C07257=1101.391,313.700,-81.925,179.212,17.147,151.820
C07258=1101.385,313.452,-81.894,179.209,17.145,151.820
C07259=1101.379,313.204,-81.863,179.206,17.143,151.820
C07260=1101.373,312.956,-81.831,179.203,17.142,151.820
C07261=1101.368,312.708,-81.800,179.200,17.140,151.820
C07262=1101.362,312.461,-81.769,179.196,17.137,151.821
C07263=1101.356,312.212,-81.737,179.193,17.135,151.821
C07264=1101.350,311.965,-81.706,179.189,17.133,151.821
C07265=1101.345,311.716,-81.675,179.186,17.131,151.821
C07266=1101.339,311.469,-81.644,179.183,17.129,151.821
C07267=1101.333,311.221,-81.613,179.179,17.128,151.822
C07268=1101.327,310.972,-81.581,179.175,17.126,151.822
C07269=1101.322,310.725,-81.550,179.172,17.124,151.822
C07270=1101.316,310.477,-81.519,179.169,17.121,151.822
C07271=1101.310,310.229,-81.488,179.165,17.119,151.822
C07272=1101.304,309.981,-81.456,179.162,17.117,151.823
C07273=1101.299,309.733,-81.425,179.158,17.115,151.823
C07274=1101.293,309.485,-81.394,179.156,17.114,151.823
C07275=1101.288,309.237,-81.363,179.152,17.112,151.823
C07276=1101.282,308.989,-81.333,179.149,17.110,151.824
C07277=1101.276,308.741,-81.301,179.145,17.108,151.824
C07278=1101.270,308.493,-81.270,179.142,17.106,151.824
C07279=1101.265,308.245,-81.239,179.138,17.104,151.824
C07280=1101.259,307.998,-81.208,179.135,17.102,151.824
C07281=1101.253,307.749,-81.177,179.131,17.100,151.825
C07282=1101.247,307.501,-81.147,179.128,17.098,151.825
C07283=1101.242,307.254,-81.115,179.124,17.096,151.825
C07284=1101.236,307.006,-81.085,179.121,17.094,151.825
C07285=1101.230,306.757,-81.053,179.118,17.093,151.826
C07286=1101.225,306.509,-81.023,179.115,17.091,151.826
C07287=1101.219,306.262,-80.991,179.111,17.089,151.826
C07288=1101.213,306.014,-80.961,179.108,17.087,151.826
C07289=1101.208,305.766,-80.930,179.104,17.085,151.826
C07290=1101.202,305.517,-80.899,179.101,17.083,151.827
C07291=1101.197,305.269,-80.868,179.097,17.081,151.827
C07292=1101.191,305.022,-80.837,179.094,17.079,151.827
C07293=1101.186,304.774,-80.806,179.090,17.078,151.827
C07294=1101.180,304.526,-80.776,179.087,17.075,151.828
C07295=1101.174,304.277,-80.745,179.084,17.074,151.828
C07296=1101.168,304.029,-80.714,179.081,17.072,151.828
C07297=1101.162,303.781,-80.684,179.077,17.070,151.828
C07298=1101.154,303.400,-80.636,179.072,17.068,151.829
C07299=1101.146,303.018,-80.589,179.067,17.065,151.829
C07300=1101.137,302.637,-80.542,179.061,17.062,151.830
C07301=1101.128,302.254,-80.495,179.056,17.059,151.830
C07302=1101.123,302.006,-80.464,179.053,17.057,151.830
C07303=1101.117,301.758,-80.433,179.049,17.055,151.830
C07304=1101.111,301.511,-80.403,179.045,17.053,151.831
C07305=1101.106,301.262,-80.373,179.042,17.051,151.831
C07306=1101.100,301.014,-80.342,179.039,17.050,151.831
C07307=1101.095,300.766,-80.312,179.036,17.048,151.831
C07308=1101.089,300.518,-80.281,179.032,17.046,151.832
C07309=1101.084,300.270,-80.251,179.029,17.044,151.832
C07310=1101.078,300.022,-80.221,179.025,17.042,151.832
C07311=1101.073,299.774,-80.190,179.022,17.040,151.832
C07312=1101.067,299.527,-80.159,179.019,17.039,151.833
C07313=1101.061,299.278,-80.130,179.015,17.037,151.833
C07314=1101.056,299.030,-80.099,179.012,17.035,151.833
C07315=1101.051,298.782,-80.068,179.008,17.034,151.834
C07316=1101.045,298.534,-80.038,179.005,17.032,151.834
C07317=1101.039,298.286,-80.008,179.001,17.030,151.834
C07318=1101.034,298.038,-79.977,178.998,17.028,151.834
C07319=1101.028,297.790,-79.947,178.995,17.027,151.835
C07320=1101.022,297.542,-79.917,178.991,17.025,151.835
C07321=1101.017,297.294,-79.886,178.988,17.023,151.835
C07322=1101.011,297.046,-79.857,178.984,17.021,151.835
C07323=1101.005,296.798,-79.826,178.981,17.019,151.836
C07324=1101.000,296.550,-79.796,178.978,17.018,151.836
C07325=1100.994,296.302,-79.766,178.974,17.016,151.836
C07326=1100.986,295.953,-79.723,178.969,17.014,151.837
C07327=1100.978,295.604,-79.681,178.964,17.012,151.837
C07328=1100.970,295.257,-79.639,178.960,17.010,151.838
C07329=1100.961,294.908,-79.596,178.954,17.007,151.838
C07330=1100.956,294.659,-79.567,178.952,17.006,151.838
C07331=1100.950,294.412,-79.536,178.948,17.004,151.839
C07332=1100.945,294.164,-79.507,178.944,17.002,151.839
C07333=1100.939,293.916,-79.477,178.941,17.000,151.839
C07334=1100.934,293.668,-79.447,178.938,16.999,151.840
C07335=1100.928,293.420,-79.417,178.934,16.997,151.840
C07336=1100.922,293.171,-79.387,178.931,16.996,151.840
C07337=1100.917,292.924,-79.357,178.927,16.994,151.841
C07338=1100.911,292.675,-79.327,178.924,16.992,151.841
C07339=1100.905,292.427,-79.297,178.921,16.991,151.841
C07340=1100.900,292.179,-79.267,178.917,16.989,151.841
C07341=1100.894,291.931,-79.237,178.914,16.987,151.842
C07342=1100.888,291.683,-79.207,178.910,16.986,151.842
C07343=1100.883,291.434,-79.178,178.907,16.985,151.842
C07344=1100.877,291.186,-79.147,178.903,16.983,151.843
C07345=1100.872,290.938,-79.118,178.900,16.981,151.843
C07346=1100.866,290.689,-79.088,178.896,16.979,151.843
C07347=1100.860,290.442,-79.058,178.893,16.978,151.844
C07348=1100.855,290.194,-79.029,178.889,16.977,151.844
C07349=1100.849,289.946,-78.999,178.886,16.975,151.844
C07350=1100.843,289.678,-78.967,178.882,16.973,151.845
C07351=1100.837,289.410,-78.935,178.879,16.972,151.845
C07352=1100.830,289.143,-78.903,178.875,16.970,151.845
C07353=1100.824,288.875,-78.871,178.871,16.968,151.846
C07354=1100.819,288.627,-78.841,178.867,16.967,151.846
C07355=1100.814,288.379,-78.812,178.864,16.965,151.846
C07356=1100.807,288.132,-78.782,178.861,16.964,151.847
C07357=1100.802,287.883,-78.752,178.857,16.963,151.847
C07358=1100.796,287.635,-78.723,178.853,16.961,151.847
C07359=1100.790,287.387,-78.694,178.851,16.960,151.848
C07360=1100.784,287.138,-78.664,178.847,16.958,151.848
C07361=1100.779,286.890,-78.634,178.843,16.957,151.849
C07362=1100.773,286.642,-78.604,178.840,16.955,151.849
C07363=1100.767,286.394,-78.575,178.837,16.954,151.849
C07364=1100.762,286.146,-78.546,178.833,16.952,151.849
C07365=1100.756,285.898,-78.516,178.829,16.950,151.850
C07366=1100.750,285.649,-78.487,178.826,16.949,151.850
C07367=1100.745,285.401,-78.457,178.823,16.948,151.851
C07368=1100.740,285.153,-78.428,178.819,16.946,151.851
C07369=1100.733,284.905,-78.399,178.815,16.945,151.851
C07370=1100.728,284.657,-78.370,178.812,16.944,151.852
C07371=1100.722,284.408,-78.340,178.809,16.942,151.852
C07372=1100.716,284.160,-78.311,178.805,16.940,151.852
C07373=1100.711,283.912,-78.282,178.801,16.939,151.853
C07374=1100.706,283.664,-78.252,178.798,16.938,151.853
C07375=1100.699,283.416,-78.223,178.795,16.936,151.853
C07376=1100.694,283.167,-78.193,178.791,16.934,151.854
C07377=1100.688,282.920,-78.165,178.788,16.933,151.854
C07378=1100.683,282.671,-78.135,178.785,16.931,151.854
C07379=1100.678,282.422,-78.106,178.781,16.930,151.855
C07380=1100.671,282.174,-78.077,178.778,16.929,151.855
C07381=1100.666,281.927,-78.048,178.774,16.927,151.856
C07382=1100.660,281.678,-78.019,178.771,16.926,151.856
C07383=1100.655,281.430,-77.989,178.768,16.925,151.856
C07384=1100.649,281.182,-77.959,178.764,16.923,151.857
C07385=1100.644,280.933,-77.931,178.760,16.921,151.857
C07386=1100.638,280.685,-77.902,178.756,16.920,151.857
C07387=1100.632,280.437,-77.873,178.754,16.919,151.858
C07388=1100.626,280.189,-77.844,178.750,16.917,151.858
C07389=1100.621,279.941,-77.815,178.746,16.916,151.859
C07390=1100.615,279.692,-77.786,178.743,16.915,151.859
C07391=1100.609,279.444,-77.757,178.739,16.913,151.859
C07392=1100.604,279.196,-77.728,178.735,16.912,151.860
C07393=1100.599,278.947,-77.699,178.733,16.911,151.860
C07394=1100.592,278.699,-77.670,178.729,16.909,151.860
C07395=1100.587,278.452,-77.641,178.725,16.908,151.861
C07396=1100.582,278.203,-77.612,178.722,16.907,151.861
C07397=1100.575,277.955,-77.583,178.718,16.905,151.862
C07398=1100.570,277.707,-77.554,178.715,16.903,151.862
C07399=1100.564,277.458,-77.526,178.712,16.902,151.862
C07400=1100.558,277.210,-77.497,178.708,16.901,151.863
C07401=1100.554,276.962,-77.468,178.704,16.900,151.863
C07402=1100.545,276.603,-77.426,178.699,16.898,151.864
C07403=1100.537,276.244,-77.384,178.695,16.896,151.864
C07404=1100.528,275.886,-77.344,178.690,16.894,151.865
C07405=1100.520,275.528,-77.302,178.684,16.892,151.865
C07406=1100.515,275.279,-77.273,178.681,16.891,151.866
C07407=1100.509,275.031,-77.244,178.677,16.890,151.866
C07408=1100.504,274.783,-77.216,178.674,16.889,151.867
C07409=1100.498,274.534,-77.187,178.671,16.887,151.867
C07410=1100.493,274.287,-77.158,178.667,16.886,151.867
C07411=1100.487,274.038,-77.130,178.664,16.885,151.868
C07412=1100.481,273.790,-77.101,178.660,16.883,151.868
C07413=1100.475,273.542,-77.073,178.656,16.882,151.869
C07414=1100.470,273.293,-77.044,178.653,16.881,151.869
C07415=1100.464,273.045,-77.015,178.650,16.879,151.869
C07416=1100.458,272.796,-76.987,178.646,16.878,151.870
C07417=1100.452,272.548,-76.958,178.643,16.877,151.870
C07418=1100.447,272.300,-76.930,178.639,16.875,151.871
C07419=1100.441,272.052,-76.902,178.636,16.875,151.871
C07420=1100.436,271.804,-76.872,178.632,16.873,151.871
C07421=1100.430,271.555,-76.844,178.628,16.872,151.872
C07422=1100.425,271.307,-76.816,178.625,16.871,151.872
C07423=1100.419,271.058,-76.788,178.622,16.869,151.873
C07424=1100.412,270.810,-76.759,178.619,16.868,151.873
C07425=1100.407,270.562,-76.731,178.615,16.867,151.874
C07426=1100.401,270.313,-76.702,178.611,16.865,151.874
C07427=1100.397,270.065,-76.674,178.608,16.864,151.874
C07428=1100.391,269.816,-76.645,178.604,16.863,151.875
C07429=1100.385,269.569,-76.617,178.601,16.862,151.875
C07430=1100.379,269.320,-76.588,178.598,16.861,151.876
C07431=1100.374,269.072,-76.561,178.594,16.860,151.876
C07432=1100.368,268.823,-76.532,178.591,16.859,151.876
C07433=1100.362,268.575,-76.504,178.587,16.857,151.877
C07434=1100.356,268.326,-76.476,178.584,16.856,151.877
C07435=1100.351,268.078,-76.448,178.580,16.855,151.878
C07436=1100.345,267.830,-76.420,178.576,16.853,151.878
C07437=1100.340,267.582,-76.391,178.573,16.853,151.879
C07438=1100.334,267.333,-76.363,178.569,16.851,151.879
C07439=1100.328,267.085,-76.335,178.566,16.850,151.879
C07440=1100.322,266.837,-76.306,178.562,16.849,151.880
C07441=1100.317,266.589,-76.278,178.559,16.847,151.880
C07442=1100.312,266.341,-76.250,178.556,16.846,151.881
C07443=1100.306,266.092,-76.222,178.552,16.845,151.881
C07444=1100.300,265.844,-76.194,178.549,16.844,151.882
C07445=1100.294,265.595,-76.166,178.545,16.843,151.882
C07446=1100.289,265.347,-76.138,178.542,16.842,151.882
C07447=1100.283,265.098,-76.110,178.538,16.840,151.883
C07448=1100.277,264.850,-76.083,178.534,16.839,151.883
C07449=1100.272,264.602,-76.055,178.531,16.838,151.884
C07450=1100.266,264.353,-76.027,178.528,16.837,151.884
C07451=1100.261,264.105,-75.999,178.524,16.836,151.885
C07452=1100.255,263.856,-75.970,178.521,16.835,151.885
C07453=1100.249,263.608,-75.942,178.517,16.834,151.886
C07454=1100.240,263.253,-75.903,178.513,16.832,151.886
C07455=1100.232,262.897,-75.863,178.507,16.830,151.887
C07456=1100.224,262.540,-75.823,178.502,16.829,151.888
C07457=1100.216,262.185,-75.784,178.497,16.827,151.888
C07458=1100.210,261.936,-75.755,178.494,16.827,151.889
C07459=1100.205,261.688,-75.727,178.490,16.825,151.889
C07460=1100.198,261.439,-75.700,178.487,16.825,151.890
C07461=1100.193,261.191,-75.672,178.483,16.823,151.890
C07462=1100.188,260.943,-75.644,178.480,16.822,151.890
C07463=1100.181,260.695,-75.617,178.476,16.821,151.891
C07464=1100.176,260.446,-75.589,178.473,16.820,151.891
C07465=1100.171,260.198,-75.561,178.469,16.819,151.892
C07466=1100.164,259.950,-75.534,178.465,16.818,151.892
C07467=1100.159,259.701,-75.506,178.462,16.817,151.893
C07468=1100.153,259.452,-75.478,178.458,16.815,151.893
C07469=1100.147,259.205,-75.451,178.455,16.815,151.894
C07470=1100.142,258.956,-75.424,178.451,16.813,151.894
C07471=1100.136,258.707,-75.395,178.448,16.813,151.895
C07472=1100.130,258.459,-75.369,178.444,16.811,151.895
C07473=1100.125,258.211,-75.341,178.441,16.811,151.896
C07474=1100.118,257.962,-75.313,178.437,16.809,151.896
C07475=1100.113,257.714,-75.286,178.434,16.809,151.896
C07476=1100.108,257.466,-75.258,178.430,16.807,151.897
C07477=1100.102,257.217,-75.231,178.427,16.806,151.897
C07478=1100.096,256.968,-75.203,178.423,16.805,151.898
C07479=1100.090,256.720,-75.176,178.420,16.804,151.898
C07480=1100.085,256.472,-75.148,178.416,16.803,151.899
C07481=1100.079,256.223,-75.120,178.413,16.802,151.899
C07482=1100.073,255.975,-75.093,178.409,16.801,151.900
C07483=1100.068,255.726,-75.066,178.406,16.800,151.900
C07484=1100.062,255.478,-75.039,178.402,16.799,151.901
C07485=1100.056,255.229,-75.011,178.399,16.798,151.901
C07486=1100.051,254.981,-74.984,178.395,16.797,151.902
C07487=1100.045,254.733,-74.956,178.392,16.796,151.902
C07488=1100.039,254.484,-74.930,178.388,16.795,151.902
C07489=1100.034,254.235,-74.902,178.385,16.794,151.903
C07490=1100.028,253.987,-74.875,178.381,16.793,151.903
C07491=1100.023,253.739,-74.847,178.378,16.792,151.904
C07492=1100.017,253.490,-74.821,178.375,16.791,151.904
C07493=1100.012,253.242,-74.793,178.371,16.790,151.905
C07494=1100.006,252.994,-74.766,178.368,16.788,151.905
C07495=1100.000,252.744,-74.739,178.364,16.788,151.906
C07496=1099.994,252.496,-74.712,178.360,16.787,151.906
C07497=1099.989,252.248,-74.684,178.357,16.786,151.907
C07498=1099.983,252.000,-74.657,178.353,16.785,151.907
C07499=1099.978,251.751,-74.630,178.350,16.784,151.908
C07500=1099.973,251.503,-74.603,178.346,16.783,151.908
C07501=1099.967,251.253,-74.576,178.344,16.782,151.908
C07502=1099.961,251.005,-74.548,178.340,16.780,151.909
C07503=1099.956,250.757,-74.521,178.337,16.779,151.909
C07504=1099.950,250.508,-74.495,178.333,16.778,151.910
C07505=1099.945,250.260,-74.467,178.329,16.778,151.910
C07506=1099.937,249.901,-74.429,178.325,16.776,151.911
C07507=1099.929,249.543,-74.389,178.319,16.775,151.912
C07508=1099.921,249.184,-74.351,178.314,16.773,151.913
C07509=1099.913,248.825,-74.312,178.310,16.772,151.913
C07510=1099.907,248.577,-74.285,178.306,16.771,151.914
C07511=1099.902,248.329,-74.258,178.303,16.770,151.914
C07512=1099.896,248.079,-74.231,178.299,16.768,151.915
C07513=1099.890,247.831,-74.204,178.295,16.768,151.915
C07514=1099.885,247.583,-74.178,178.292,16.766,151.915
C07515=1099.879,247.334,-74.150,178.288,16.766,151.916
C07516=1099.874,247.086,-74.124,178.285,16.764,151.916
C07517=1099.868,246.837,-74.097,178.282,16.764,151.917
C07518=1099.862,246.589,-74.070,178.278,16.763,151.917
C07519=1099.857,246.340,-74.043,178.275,16.762,151.918
C07520=1099.851,246.092,-74.016,178.271,16.761,151.918
C07521=1099.846,245.843,-73.990,178.267,16.760,151.919
C07522=1099.840,245.595,-73.963,178.264,16.759,151.919
C07523=1099.835,245.346,-73.936,178.260,16.758,151.920
C07524=1099.829,245.098,-73.909,178.257,16.757,151.920
C07525=1099.823,244.850,-73.883,178.253,16.756,151.921
C07526=1099.818,244.601,-73.857,178.250,16.755,151.921
C07527=1099.812,244.352,-73.830,178.246,16.754,151.922
C07528=1099.807,244.104,-73.803,178.243,16.753,151.922
C07529=1099.801,243.855,-73.776,178.240,16.753,151.923
C07530=1099.795,243.607,-73.750,178.236,16.752,151.923
C07531=1099.790,243.358,-73.724,178.233,16.751,151.924
C07532=1099.784,243.110,-73.697,178.229,16.750,151.924
C07533=1099.778,242.861,-73.670,178.226,16.749,151.925
C07534=1099.773,242.613,-73.644,178.222,16.747,151.925
C07535=1099.767,242.364,-73.618,178.219,16.747,151.926
C07536=1099.761,242.116,-73.591,178.216,16.746,151.926
C07537=1099.756,241.867,-73.564,178.212,16.745,151.927
C07538=1099.750,241.619,-73.538,178.208,16.745,151.927
C07539=1099.744,241.370,-73.512,178.205,16.743,151.928
C07540=1099.739,241.122,-73.485,178.201,16.743,151.928
C07541=1099.733,240.873,-73.459,178.198,16.742,151.929
C07542=1099.727,240.624,-73.433,178.194,16.741,151.929
C07543=1099.722,240.376,-73.406,178.191,16.740,151.930
C07544=1099.716,240.127,-73.380,178.187,16.739,151.930
C07545=1099.710,239.878,-73.353,178.184,16.738,151.931
C07546=1099.705,239.630,-73.327,178.180,16.737,151.931
C07547=1099.699,239.381,-73.301,178.177,16.736,151.932
C07548=1099.693,239.133,-73.274,178.174,16.736,151.932
C07549=1099.688,238.884,-73.248,178.170,16.735,151.933
C07550=1099.682,238.635,-73.222,178.167,16.734,151.933
C07551=1099.677,238.386,-73.196,178.163,16.733,151.934
C07552=1099.671,238.138,-73.169,178.160,16.732,151.934
C07553=1099.665,237.889,-73.143,178.156,16.732,151.935
C07554=1099.660,237.641,-73.116,178.152,16.731,151.935
C07555=1099.654,237.392,-73.090,178.149,16.730,151.936
C07556=1099.649,237.144,-73.064,178.145,16.728,151.936
C07557=1099.643,236.895,-73.039,178.142,16.728,151.937
C07558=1099.634,236.529,-72.999,178.137,16.727,151.938
C07559=1099.626,236.164,-72.961,178.132,16.725,151.938
C07560=1099.618,235.798,-72.923,178.127,16.724,151.939
C07561=1099.610,235.433,-72.885,178.122,16.723,151.940
C07562=1099.604,235.184,-72.859,178.119,16.722,151.940
C07563=1099.598,234.936,-72.832,178.115,16.721,151.941
C07564=1099.593,234.688,-72.807,178.111,16.721,151.941
C07565=1099.587,234.439,-72.781,178.108,16.720,151.942
C07566=1099.582,234.191,-72.754,178.104,16.719,151.942
C07567=1099.576,233.942,-72.729,178.101,16.718,151.943
C07568=1099.571,233.693,-72.703,178.098,16.718,151.943
C07569=1099.564,233.444,-72.677,178.094,16.716,151.944
C07570=1099.559,233.196,-72.651,178.091,16.716,151.944
C07571=1099.554,232.947,-72.625,178.087,16.714,151.945
C07572=1099.548,232.698,-72.599,178.084,16.714,151.945
C07573=1099.542,232.450,-72.574,178.081,16.713,151.946
C07574=1099.536,232.201,-72.547,178.077,16.712,151.946
C07575=1099.532,231.953,-72.522,178.074,16.711,151.947
C07576=1099.525,231.704,-72.496,178.070,16.711,151.948
C07577=1099.520,231.455,-72.470,178.066,16.710,151.948
C07578=1099.514,231.206,-72.444,178.063,16.709,151.949
C07579=1099.509,230.959,-72.418,178.060,16.708,151.949
C07580=1099.503,230.710,-72.393,178.056,16.707,151.950
C07581=1099.498,230.461,-72.367,178.053,16.707,151.950
C07582=1099.491,230.212,-72.341,178.050,16.706,151.951
C07583=1099.486,229.963,-72.316,178.046,16.705,151.951
C07584=1099.481,229.715,-72.290,178.042,16.705,151.952
C07585=1099.475,229.467,-72.265,178.039,16.704,151.952
C07586=1099.469,229.218,-72.239,178.035,16.703,151.953
C07587=1099.463,228.969,-72.213,178.032,16.702,151.953
C07588=1099.458,228.721,-72.188,178.029,16.702,151.954
C07589=1099.452,228.472,-72.162,178.025,16.700,151.954
C07590=1099.447,228.223,-72.137,178.022,16.700,151.955
C07591=1099.440,227.974,-72.111,178.018,16.699,151.955
C07592=1099.436,227.726,-72.086,178.014,16.698,151.956
C07593=1099.429,227.477,-72.060,178.011,16.698,151.956
C07594=1099.424,227.228,-72.034,178.008,16.697,151.957
C07595=1099.418,226.980,-72.009,178.004,16.696,151.957
C07596=1099.413,226.731,-71.983,178.001,16.695,151.958
C07597=1099.407,226.483,-71.958,177.998,16.695,151.959
C07598=1099.401,226.234,-71.932,177.994,16.694,151.959
C07599=1099.395,225.986,-71.907,177.991,16.693,151.960
C07600=1099.390,225.737,-71.881,177.987,16.693,151.960
C07601=1099.384,225.488,-71.856,177.983,16.692,151.961
C07602=1099.379,225.240,-71.830,177.980,16.691,151.961
C07603=1099.373,224.991,-71.806,177.977,16.690,151.962
C07604=1099.368,224.742,-71.780,177.973,16.689,151.962
C07605=1099.362,224.494,-71.755,177.970,16.689,151.963
C07606=1099.356,224.245,-71.729,177.967,16.688,151.963
C07607=1099.351,223.997,-71.704,177.963,16.687,151.964
C07608=1099.346,223.747,-71.679,177.960,16.686,151.964
C07609=1099.340,223.498,-71.653,177.956,16.686,151.965
C07610=1099.331,223.125,-71.616,177.951,16.685,151.966
C07611=1099.323,222.751,-71.578,177.946,16.683,151.966
C07612=1099.314,222.377,-71.540,177.941,16.682,151.967
C07613=1099.306,222.003,-71.502,177.936,16.681,151.968
C07614=1099.300,221.754,-71.477,177.932,16.680,151.968
C07615=1099.295,221.506,-71.452,177.928,16.679,151.969
C07616=1099.289,221.257,-71.426,177.925,16.679,151.970
C07617=1099.283,221.008,-71.401,177.922,16.678,151.970
C07618=1099.278,220.760,-71.376,177.919,16.678,151.971
C07619=1099.272,220.510,-71.351,177.915,16.677,151.971
C07620=1099.266,220.261,-71.325,177.911,16.676,151.972
C07621=1099.261,220.014,-71.300,177.908,16.676,151.972
C07622=1099.255,219.764,-71.276,177.904,16.675,151.973
C07623=1099.249,219.516,-71.251,177.901,16.674,151.973
C07624=1099.243,219.267,-71.226,177.898,16.674,151.974
C07625=1099.238,219.019,-71.201,177.895,16.673,151.975
C07626=1099.232,218.770,-71.175,177.890,16.672,151.975
C07627=1099.227,218.521,-71.151,177.888,16.671,151.976
C07628=1099.221,218.273,-71.126,177.884,16.671,151.976
C07629=1099.215,218.023,-71.101,177.880,16.670,151.977
C07630=1099.210,217.775,-71.076,177.877,16.669,151.977
C07631=1099.204,217.526,-71.051,177.874,16.669,151.978
C07632=1099.198,217.278,-71.026,177.871,16.668,151.978
C07633=1099.193,217.029,-71.001,177.867,16.667,151.979
C07634=1099.187,216.780,-70.977,177.863,16.667,151.979
C07635=1099.182,216.531,-70.951,177.860,16.666,151.980
C07636=1099.177,216.282,-70.927,177.857,16.666,151.980
C07637=1099.170,216.034,-70.902,177.853,16.665,151.981
C07638=1099.165,215.785,-70.877,177.850,16.664,151.981
C07639=1099.159,215.536,-70.853,177.847,16.663,151.982
C07640=1099.153,215.288,-70.828,177.843,16.663,151.983
C07641=1099.148,215.039,-70.803,177.839,16.662,151.983
C07642=1099.142,214.790,-70.779,177.836,16.661,151.984
C07643=1099.137,214.542,-70.753,177.833,16.661,151.984
C07644=1099.132,214.293,-70.729,177.830,16.660,151.985
C07645=1099.126,214.044,-70.704,177.826,16.659,151.985
C07646=1099.120,213.795,-70.679,177.822,16.659,151.986
C07647=1099.115,213.547,-70.655,177.819,16.658,151.986
C07648=1099.109,213.298,-70.631,177.816,16.657,151.987
C07649=1099.103,213.049,-70.605,177.812,16.656,151.987
C07650=1099.098,212.801,-70.581,177.809,16.656,151.988
C07651=1099.092,212.552,-70.556,177.806,16.655,151.988
C07652=1099.087,212.303,-70.532,177.802,16.655,151.989
C07653=1099.081,212.054,-70.507,177.798,16.654,151.990
C07654=1099.075,211.806,-70.482,177.795,16.653,151.990
C07655=1099.070,211.557,-70.458,177.792,16.653,151.991
C07656=1099.064,211.308,-70.434,177.789,16.652,151.991
C07657=1099.059,211.059,-70.409,177.785,16.651,151.992
C07658=1099.053,210.810,-70.385,177.781,16.651,151.992
C07659=1099.047,210.562,-70.360,177.778,16.650,151.993
C07660=1099.042,210.313,-70.336,177.775,16.650,151.993
C07661=1099.035,210.064,-70.311,177.772,16.649,151.994
C07662=1099.028,209.694,-70.275,177.767,16.648,151.995
C07663=1099.019,209.324,-70.239,177.761,16.647,151.995
C07664=1099.010,208.954,-70.202,177.756,16.646,151.996
C07665=1099.002,208.584,-70.166,177.751,16.645,151.997
C07666=1098.979,207.575,-70.068,177.709,16.631,152.003
C07667=1098.974,207.326,-70.044,177.705,16.631,152.003
C07668=1098.968,207.078,-70.020,177.702,16.632,152.004
C07669=1098.963,206.829,-69.997,177.698,16.632,152.005
C07670=1098.957,206.579,-69.972,177.694,16.632,152.006
C07671=1098.951,206.331,-69.948,177.691,16.632,152.007
C07672=1098.945,206.082,-69.924,177.687,16.632,152.007
C07673=1098.940,205.834,-69.900,177.683,16.632,152.008
C07674=1098.934,205.585,-69.876,177.680,16.632,152.009
C07675=1098.928,205.336,-69.853,177.676,16.633,152.010
C07676=1098.923,205.087,-69.828,177.673,16.633,152.010
C07677=1098.918,204.839,-69.804,177.670,16.633,152.011
C07678=1098.911,204.590,-69.780,177.666,16.634,152.012
C07679=1098.906,204.340,-69.756,177.662,16.634,152.013
C07680=1098.901,204.092,-69.732,177.658,16.634,152.014
C07681=1098.895,203.843,-69.709,177.655,16.634,152.014
C07682=1098.890,203.594,-69.685,177.651,16.634,152.015
C07683=1098.883,203.345,-69.661,177.648,16.635,152.016
C07684=1098.878,203.097,-69.637,177.644,16.635,152.017
C07685=1098.873,202.848,-69.613,177.640,16.635,152.017
C07686=1098.867,202.599,-69.590,177.637,16.635,152.018
C07687=1098.862,202.351,-69.565,177.633,16.635,152.019
C07688=1098.855,202.101,-69.542,177.630,16.636,152.020
C07689=1098.850,201.852,-69.518,177.627,16.636,152.020
C07690=1098.844,201.604,-69.494,177.623,16.636,152.021
C07691=1098.838,201.355,-69.471,177.619,16.637,152.022
C07692=1098.832,201.106,-69.446,177.616,16.637,152.023
C07693=1098.826,200.858,-69.423,177.612,16.637,152.024
C07694=1098.821,200.609,-69.399,177.608,16.637,152.024
C07695=1098.815,200.360,-69.376,177.605,16.637,152.025
C07696=1098.810,200.111,-69.352,177.601,16.638,152.026
C07697=1098.804,199.862,-69.328,177.598,16.638,152.027
C07698=1098.798,199.613,-69.305,177.594,16.639,152.027
C07699=1098.793,199.365,-69.281,177.591,16.639,152.028
C07700=1098.787,199.116,-69.258,177.587,16.639,152.029
C07701=1098.781,198.867,-69.234,177.583,16.639,152.030
C07702=1098.776,198.618,-69.211,177.580,16.639,152.030
C07703=1098.769,198.369,-69.187,177.576,16.639,152.031
C07704=1098.764,198.120,-69.163,177.573,16.639,152.032
C07705=1098.758,197.872,-69.139,177.569,16.639,152.033
C07706=1098.752,197.623,-69.117,177.566,16.640,152.033
C07707=1098.747,197.374,-69.092,177.562,16.641,152.034
C07708=1098.741,197.125,-69.069,177.559,16.641,152.035
C07709=1098.736,196.876,-69.046,177.555,16.641,152.036
C07710=1098.730,196.628,-69.022,177.552,16.641,152.036
C07711=1098.725,196.379,-68.999,177.548,16.641,152.037
C07712=1098.718,196.129,-68.976,177.544,16.641,152.038
C07713=1098.713,195.881,-68.952,177.541,16.641,152.039
C07714=1098.707,195.632,-68.929,177.537,16.641,152.039
C07715=1098.701,195.383,-68.906,177.534,16.642,152.040
C07716=1098.696,195.134,-68.881,177.531,16.642,152.041
C07717=1098.690,194.885,-68.859,177.527,16.642,152.042
C07718=1098.685,194.637,-68.836,177.524,16.642,152.042
C07719=1098.679,194.388,-68.812,177.520,16.643,152.043
C07720=1098.674,194.139,-68.788,177.516,16.643,152.044
C07721=1098.668,193.890,-68.765,177.513,16.643,152.045
C07722=1098.662,193.641,-68.742,177.509,16.643,152.045
C07723=1098.657,193.393,-68.718,177.507,16.643,152.046
C07724=1098.651,193.144,-68.695,177.503,16.643,152.047
C07725=1098.645,192.895,-68.672,177.499,16.644,152.048
C07726=1098.640,192.646,-68.649,177.496,16.644,152.048
C07727=1098.633,192.373,-68.623,177.492,16.644,152.049
C07728=1098.627,192.099,-68.598,177.488,16.644,152.050
C07729=1098.621,191.825,-68.572,177.485,16.644,152.051
C07730=1098.615,191.552,-68.547,177.480,16.644,152.052
C07731=1098.610,191.303,-68.524,177.477,16.645,152.052
C07732=1098.604,191.054,-68.501,177.474,16.645,152.053
C07733=1098.599,190.805,-68.478,177.470,16.645,152.054
C07734=1098.593,190.557,-68.454,177.467,16.645,152.054
C07735=1098.588,190.307,-68.431,177.463,16.645,152.055
C07736=1098.582,190.058,-68.408,177.460,16.645,152.056
C07737=1098.576,189.810,-68.385,177.456,16.645,152.057
C07738=1098.570,189.561,-68.362,177.452,16.645,152.058
C07739=1098.565,189.312,-68.339,177.450,16.646,152.058
C07740=1098.560,189.063,-68.315,177.446,16.646,152.059
C07741=1098.554,188.814,-68.292,177.442,16.646,152.060
C07742=1098.548,188.565,-68.269,177.439,16.646,152.060
C07743=1098.543,188.316,-68.247,177.435,16.646,152.061
C07744=1098.537,188.068,-68.224,177.432,16.646,152.062
C07745=1098.532,187.819,-68.201,177.428,16.646,152.062
C07746=1098.526,187.570,-68.178,177.426,16.646,152.063
C07747=1098.521,187.321,-68.155,177.422,16.646,152.064
C07748=1098.515,187.072,-68.132,177.418,16.646,152.065
C07749=1098.509,186.823,-68.109,177.415,16.647,152.065
C07750=1098.504,186.574,-68.086,177.411,16.647,152.066
C07751=1098.498,186.325,-68.063,177.408,16.647,152.067
C07752=1098.493,186.076,-68.041,177.405,16.647,152.067
C07753=1098.487,185.827,-68.018,177.402,16.647,152.068
C07754=1098.482,185.578,-67.994,177.398,16.647,152.069
C07755=1098.477,185.329,-67.971,177.395,16.647,152.069
C07756=1098.471,185.080,-67.948,177.391,16.647,152.070
C07757=1098.465,184.832,-67.926,177.388,16.647,152.071
C07758=1098.459,184.583,-67.903,177.384,16.647,152.072
C07759=1098.453,184.333,-67.881,177.381,16.648,152.072
C07760=1098.448,184.084,-67.858,177.378,16.648,152.073
C07761=1098.443,183.836,-67.835,177.374,16.648,152.074
C07762=1098.437,183.587,-67.812,177.370,16.648,152.075
C07763=1098.430,183.339,-67.790,177.367,16.648,152.075
C07764=1098.425,183.090,-67.767,177.364,16.649,152.076
C07765=1098.419,182.840,-67.745,177.361,16.649,152.077
C07766=1098.413,182.591,-67.722,177.357,16.649,152.077
C07767=1098.408,182.343,-67.699,177.354,16.649,152.078
C07768=1098.401,182.094,-67.677,177.350,16.649,152.079
C07769=1098.396,181.844,-67.654,177.346,16.649,152.080
C07770=1098.390,181.596,-67.632,177.344,16.649,152.080
C07771=1098.385,181.347,-67.609,177.340,16.649,152.081
C07772=1098.379,181.098,-67.587,177.337,16.649,152.082
C07773=1098.373,180.849,-67.564,177.333,16.650,152.082
C07774=1098.367,180.600,-67.541,177.330,16.650,152.083
C07775=1098.362,180.351,-67.519,177.327,16.650,152.084
C07776=1098.355,180.102,-67.497,177.323,16.650,152.085
C07777=1098.350,179.853,-67.474,177.320,16.650,152.085
C07778=1098.345,179.605,-67.452,177.316,16.650,152.086
C07779=1098.339,179.356,-67.429,177.313,16.650,152.087
C07780=1098.333,179.107,-67.407,177.309,16.650,152.087
C07781=1098.327,178.858,-67.385,177.306,16.651,152.088
C07782=1098.322,178.609,-67.362,177.303,16.651,152.089
C07783=1098.317,178.360,-67.340,177.299,16.651,152.090
C07784=1098.310,178.111,-67.317,177.296,16.651,152.090
C07785=1098.305,177.862,-67.295,177.292,16.651,152.091
C07786=1098.299,177.613,-67.272,177.290,16.651,152.092
C07787=1098.293,177.364,-67.251,177.286,16.651,152.092
C07788=1098.288,177.115,-67.228,177.283,16.651,152.093
C07789=1098.282,176.866,-67.206,177.279,16.651,152.094
C07790=1098.276,176.617,-67.183,177.276,16.651,152.094
C07791=1098.270,176.343,-67.159,177.272,16.651,152.095
C07792=1098.264,176.070,-67.135,177.268,16.651,152.096
C07793=1098.258,175.795,-67.110,177.265,16.652,152.097
C07794=1098.251,175.521,-67.085,177.261,16.652,152.098
C07795=1098.246,175.272,-67.063,177.258,16.652,152.098
C07796=1098.240,175.024,-67.041,177.254,16.652,152.099
C07797=1098.234,174.774,-67.019,177.252,16.652,152.100
C07798=1098.229,174.525,-66.996,177.248,16.652,152.100
C07799=1098.224,174.277,-66.974,177.244,16.652,152.101
C07800=1098.218,174.027,-66.952,177.241,16.652,152.102
C07801=1098.212,173.779,-66.930,177.238,16.652,152.102
C07802=1098.206,173.530,-66.908,177.235,16.653,152.103
C07803=1098.201,173.281,-66.886,177.231,16.653,152.104
C07804=1098.195,173.032,-66.863,177.228,16.652,152.104
C07805=1098.190,172.783,-66.842,177.225,16.652,152.105
C07806=1098.184,172.534,-66.820,177.221,16.652,152.106
C07807=1098.178,172.285,-66.797,177.219,16.653,152.106
C07808=1098.173,172.036,-66.775,177.215,16.653,152.107
C07809=1098.167,171.787,-66.753,177.211,16.653,152.108
C07810=1098.161,171.538,-66.731,177.208,16.653,152.108
C07811=1098.156,171.289,-66.709,177.205,16.653,152.109
C07812=1098.150,171.040,-66.687,177.202,16.653,152.110
C07813=1098.145,170.791,-66.665,177.198,16.653,152.110
C07814=1098.139,170.542,-66.644,177.195,16.653,152.111
C07815=1098.133,170.293,-66.621,177.192,16.653,152.112
C07816=1098.128,170.045,-66.600,177.189,16.653,152.112
C07817=1098.122,169.795,-66.577,177.186,16.653,152.113
C07818=1098.117,169.546,-66.555,177.182,16.653,152.114
C07819=1098.111,169.297,-66.534,177.179,16.652,152.114
C07820=1098.106,169.048,-66.511,177.175,16.653,152.115
C07821=1098.100,168.800,-66.490,177.173,16.653,152.115
C07822=1098.095,168.550,-66.467,177.169,16.653,152.116
C07823=1098.089,168.302,-66.446,177.166,16.653,152.117
C07824=1098.084,168.052,-66.424,177.162,16.652,152.117
C07825=1098.078,167.804,-66.403,177.160,16.653,152.118
C07826=1098.073,167.554,-66.380,177.156,16.653,152.119
C07827=1098.067,167.306,-66.359,177.153,16.653,152.119
C07828=1098.062,167.056,-66.337,177.150,16.652,152.120
C07829=1098.055,166.807,-66.315,177.146,16.652,152.121
C07830=1098.051,166.558,-66.293,177.144,16.653,152.121
C07831=1098.044,166.309,-66.272,177.140,16.653,152.122
C07832=1098.040,166.060,-66.250,177.137,16.652,152.123
C07833=1098.033,165.811,-66.228,177.133,16.652,152.123
C07834=1098.028,165.562,-66.207,177.131,16.652,152.124
C07835=1098.022,165.313,-66.185,177.127,16.652,152.125
C07836=1098.017,165.064,-66.163,177.124,16.652,152.125
C07837=1098.012,164.816,-66.142,177.120,16.652,152.126
C07838=1098.006,164.566,-66.120,177.117,16.652,152.126
C07839=1098.001,164.318,-66.098,177.115,16.652,152.127
C07840=1097.995,164.068,-66.076,177.111,16.652,152.128
C07841=1097.990,163.820,-66.055,177.108,16.652,152.128
C07842=1097.984,163.570,-66.033,177.104,16.652,152.129
C07843=1097.978,163.322,-66.012,177.102,16.652,152.130
C07844=1097.973,163.072,-65.989,177.099,16.651,152.130
C07845=1097.967,162.824,-65.968,177.095,16.651,152.131
C07846=1097.963,162.575,-65.946,177.092,16.651,152.131
C07847=1097.957,162.325,-65.925,177.088,16.651,152.132
C07848=1097.951,162.077,-65.904,177.086,16.651,152.133
C07849=1097.946,161.827,-65.882,177.083,16.651,152.133
C07850=1097.940,161.579,-65.861,177.079,16.651,152.134
C07851=1097.934,161.329,-65.839,177.076,16.651,152.135
C07852=1097.929,161.081,-65.817,177.073,16.651,152.135
C07853=1097.923,160.831,-65.796,177.070,16.651,152.136
C07854=1097.918,160.582,-65.775,177.067,16.650,152.136
C07855=1097.911,160.308,-65.751,177.063,16.651,152.137
C07856=1097.905,160.034,-65.728,177.059,16.651,152.138
C07857=1097.899,159.759,-65.704,177.056,16.651,152.139
C07858=1097.892,159.485,-65.680,177.052,16.651,152.139
C07859=1097.887,159.236,-65.660,177.049,16.650,152.140
C07860=1097.881,158.987,-65.638,177.047,16.651,152.140
C07861=1097.875,158.738,-65.617,177.043,16.651,152.141
C07862=1097.871,158.489,-65.596,177.040,16.650,152.142
C07863=1097.865,158.239,-65.574,177.036,16.650,152.142
C07864=1097.859,157.991,-65.553,177.034,16.650,152.143
C07865=1097.853,157.741,-65.532,177.031,16.650,152.144
C07866=1097.848,157.493,-65.511,177.027,16.650,152.144
C07867=1097.842,157.244,-65.489,177.024,16.650,152.145
C07868=1097.836,156.994,-65.468,177.021,16.650,152.145
C07869=1097.831,156.746,-65.447,177.018,16.650,152.146
C07870=1097.825,156.496,-65.425,177.015,16.650,152.147
C07871=1097.820,156.247,-65.404,177.011,16.649,152.147
C07872=1097.814,155.999,-65.383,177.009,16.649,152.148
C07873=1097.809,155.749,-65.362,177.005,16.649,152.148
C07874=1097.803,155.500,-65.341,177.002,16.649,152.149
C07875=1097.797,155.251,-65.319,176.999,16.649,152.150
C07876=1097.792,155.002,-65.299,176.996,16.649,152.150
C07877=1097.786,154.753,-65.277,176.993,16.649,152.151
C07878=1097.780,154.504,-65.257,176.989,16.649,152.151
C07879=1097.775,154.255,-65.235,176.987,16.649,152.152
C07880=1097.769,154.006,-65.215,176.983,16.649,152.153
C07881=1097.763,153.757,-65.193,176.980,16.648,152.153
C07882=1097.758,153.508,-65.173,176.977,16.648,152.154
C07883=1097.752,153.259,-65.151,176.974,16.649,152.155
C07884=1097.747,153.009,-65.130,176.971,16.648,152.155
C07885=1097.741,152.761,-65.109,176.968,16.648,152.156
C07886=1097.736,152.512,-65.088,176.964,16.648,152.156
C07887=1097.730,152.263,-65.067,176.962,16.648,152.157
C07888=1097.724,152.013,-65.046,176.958,16.648,152.158
C07889=1097.719,151.764,-65.026,176.955,16.647,152.158
C07890=1097.712,151.515,-65.005,176.953,16.648,152.159
C07891=1097.707,151.266,-64.984,176.949,16.647,152.159
C07892=1097.701,151.018,-64.963,176.946,16.647,152.160
C07893=1097.696,150.769,-64.942,176.943,16.647,152.160
C07894=1097.690,150.519,-64.921,176.940,16.647,152.161
C07895=1097.685,150.270,-64.900,176.937,16.647,152.162
C07896=1097.679,150.021,-64.880,176.934,16.646,152.162
C07897=1097.674,149.771,-64.859,176.931,16.647,152.163
C07898=1097.668,149.523,-64.837,176.928,16.646,152.163
C07899=1097.663,149.274,-64.817,176.925,16.646,152.164
C07900=1097.657,149.025,-64.797,176.921,16.645,152.165
C07901=1097.651,148.776,-64.775,176.919,16.646,152.165
C07902=1097.645,148.527,-64.755,176.915,16.646,152.166
C07903=1097.640,148.277,-64.734,176.912,16.645,152.166
C07904=1097.635,148.029,-64.713,176.910,16.646,152.167
C07905=1097.628,147.779,-64.693,176.906,16.645,152.167
C07906=1097.623,147.530,-64.672,176.903,16.645,152.168
C07907=1097.617,147.281,-64.651,176.900,16.644,152.169
C07908=1097.612,147.033,-64.630,176.897,16.645,152.169
C07909=1097.605,146.783,-64.610,176.894,16.644,152.170
C07910=1097.600,146.534,-64.589,176.891,16.644,152.170
C07911=1097.595,146.285,-64.569,176.888,16.645,152.171
C07912=1097.589,146.036,-64.548,176.885,16.644,152.172
C07913=1097.583,145.787,-64.527,176.882,16.644,152.172
C07914=1097.577,145.538,-64.507,176.878,16.643,152.173
C07915=1097.572,145.289,-64.486,176.876,16.644,152.173
C07916=1097.567,145.040,-64.465,176.873,16.643,152.174
C07917=1097.561,144.791,-64.446,176.869,16.643,152.174
C07918=1097.555,144.541,-64.425,176.867,16.643,152.175
C07919=1097.549,144.267,-64.402,176.864,16.643,152.176
C07920=1097.542,143.992,-64.379,176.860,16.643,152.176
C07921=1097.537,143.718,-64.356,176.857,16.642,152.177
C07922=1097.530,143.442,-64.334,176.854,16.642,152.177
C07923=1097.525,143.193,-64.314,176.850,16.642,152.178
C07924=1097.519,142.944,-64.293,176.847,16.641,152.179
C07925=1097.513,142.695,-64.273,176.845,16.642,152.179
C07926=1097.508,142.446,-64.253,176.841,16.641,152.180
C07927=1097.503,142.197,-64.232,176.838,16.641,152.180
C07928=1097.497,141.949,-64.211,176.836,16.641,152.181
C07929=1097.491,141.699,-64.191,176.832,16.641,152.181
C07930=1097.485,141.450,-64.170,176.829,16.640,152.182
C07931=1097.480,141.200,-64.151,176.827,16.640,152.183
C07932=1097.474,140.951,-64.130,176.824,16.640,152.183
C07933=1097.469,140.703,-64.110,176.820,16.639,152.184
C07934=1097.463,140.453,-64.090,176.817,16.639,152.184
C07935=1097.458,140.204,-64.069,176.815,16.639,152.185
C07936=1097.452,139.955,-64.049,176.811,16.639,152.185
C07937=1097.446,139.706,-64.028,176.808,16.638,152.186
C07938=1097.440,139.457,-64.008,176.806,16.639,152.186
C07939=1097.435,139.208,-63.988,176.802,16.638,152.187
C07940=1097.429,138.959,-63.968,176.799,16.638,152.187
C07941=1097.424,138.710,-63.947,176.797,16.638,152.188
C07942=1097.418,138.461,-63.927,176.794,16.637,152.188
C07943=1097.412,138.212,-63.907,176.790,16.637,152.189
C07944=1097.407,137.962,-63.887,176.788,16.637,152.190
C07945=1097.401,137.713,-63.867,176.785,16.637,152.190
C07946=1097.395,137.464,-63.847,176.781,16.636,152.191
C07947=1097.390,137.215,-63.826,176.779,16.637,152.191
C07948=1097.384,136.966,-63.806,176.776,16.636,152.192
C07949=1097.378,136.717,-63.786,176.773,16.635,152.192
C07950=1097.373,136.467,-63.766,176.770,16.636,152.193
C07951=1097.367,136.218,-63.746,176.767,16.635,152.193
C07952=1097.361,135.969,-63.726,176.764,16.635,152.194
C07953=1097.355,135.721,-63.706,176.762,16.635,152.194
C07954=1097.350,135.471,-63.686,176.758,16.634,152.195
C07955=1097.344,135.222,-63.666,176.755,16.634,152.196
C07956=1097.339,134.973,-63.645,176.753,16.634,152.196
C07957=1097.333,134.724,-63.626,176.750,16.633,152.196
C07958=1097.328,134.474,-63.606,176.746,16.633,152.197
C07959=1097.322,134.225,-63.586,176.744,16.633,152.198
C07960=1097.316,133.977,-63.566,176.741,16.633,152.198
C07961=1097.311,133.727,-63.546,176.738,16.632,152.199
C07962=1097.305,133.478,-63.526,176.735,16.632,152.199
C07963=1097.300,133.229,-63.505,176.732,16.632,152.200
C07964=1097.294,132.980,-63.486,176.729,16.631,152.200
C07965=1097.288,132.731,-63.466,176.726,16.631,152.201
C07966=1097.283,132.482,-63.446,176.723,16.631,152.201
C07967=1097.277,132.232,-63.426,176.720,16.630,152.202
C07968=1097.271,131.983,-63.406,176.718,16.630,152.202
C07969=1097.265,131.735,-63.386,176.715,16.630,152.203
C07970=1097.261,131.485,-63.367,176.711,16.629,152.203
C07971=1097.255,131.236,-63.347,176.709,16.629,152.204
C07972=1097.249,130.987,-63.327,176.706,16.629,152.204
C07973=1097.243,130.738,-63.308,176.703,16.628,152.205
C07974=1097.237,130.488,-63.288,176.700,16.629,152.205
C07975=1097.232,130.239,-63.268,176.697,16.628,152.206
C07976=1097.226,129.990,-63.248,176.694,16.628,152.206
C07977=1097.220,129.741,-63.229,176.691,16.628,152.207
C07978=1097.214,129.492,-63.209,176.688,16.627,152.207
C07979=1097.209,129.243,-63.189,176.685,16.627,152.208
C07980=1097.203,128.994,-63.169,176.683,16.627,152.209
C07981=1097.198,128.744,-63.150,176.680,16.626,152.209
C07982=1097.192,128.495,-63.130,176.676,16.626,152.210
C07983=1097.185,128.221,-63.108,176.674,16.626,152.210
C07984=1097.179,127.945,-63.086,176.671,16.625,152.211
C07985=1097.173,127.671,-63.065,176.667,16.625,152.211
C07986=1097.167,127.396,-63.043,176.664,16.625,152.212
C07987=1097.161,127.147,-63.024,176.661,16.624,152.212
C07988=1097.155,126.898,-63.004,176.658,16.624,152.213
C07989=1097.149,126.649,-62.985,176.656,16.623,152.213
C07990=1097.144,126.399,-62.965,176.652,16.623,152.214
C07991=1097.138,126.150,-62.945,176.650,16.623,152.214
C07992=1097.133,125.901,-62.925,176.647,16.622,152.215
C07993=1097.127,125.651,-62.906,176.644,16.622,152.215
C07994=1097.121,125.402,-62.886,176.642,16.622,152.216
C07995=1097.115,125.153,-62.867,176.639,16.621,152.216
C07996=1097.110,124.904,-62.848,176.635,16.621,152.217
C07997=1097.104,124.655,-62.828,176.633,16.621,152.217
C07998=1097.098,124.406,-62.809,176.630,16.620,152.218
C07999=1097.093,124.157,-62.790,176.627,16.619,152.218
C08000=1097.087,123.908,-62.770,176.624,16.619,152.219
C08001=1097.081,123.658,-62.751,176.621,16.619,152.219
C08002=1097.075,123.409,-62.731,176.619,16.619,152.220
C08003=1097.071,123.160,-62.711,176.616,16.618,152.220
C08004=1097.065,122.911,-62.692,176.613,16.618,152.221
C08005=1097.059,122.662,-62.673,176.611,16.617,152.221
C08006=1097.054,122.412,-62.653,176.607,16.617,152.222
C08007=1097.048,122.163,-62.633,176.604,16.616,152.222
C08008=1097.042,121.914,-62.614,176.602,16.616,152.223
C08009=1097.037,121.665,-62.595,176.599,16.616,152.223
C08010=1097.031,121.416,-62.576,176.596,16.615,152.224
C08011=1097.026,121.166,-62.557,176.593,16.615,152.224
C08012=1097.020,120.917,-62.538,176.591,16.614,152.224
C08013=1097.014,120.668,-62.518,176.588,16.614,152.225
C08014=1097.009,120.419,-62.499,176.585,16.614,152.225
C08015=1097.003,120.170,-62.479,176.582,16.613,152.226
C08016=1096.997,119.920,-62.460,176.580,16.613,152.226
C08017=1096.992,119.671,-62.441,176.577,16.612,152.227
C08018=1096.986,119.422,-62.422,176.574,16.611,152.227
C08019=1096.981,119.173,-62.403,176.571,16.611,152.228
C08020=1096.975,118.924,-62.383,176.568,16.611,152.228
C08021=1096.969,118.675,-62.364,176.566,16.611,152.229
C08022=1096.964,118.425,-62.344,176.563,16.610,152.229
C08023=1096.958,118.176,-62.326,176.560,16.609,152.229
C08024=1096.953,117.927,-62.306,176.558,16.609,152.230
C08025=1096.947,117.678,-62.287,176.555,16.608,152.230
C08026=1096.942,117.429,-62.268,176.552,16.608,152.231
C08027=1096.936,117.179,-62.249,176.549,16.608,152.231
C08028=1096.931,116.930,-62.230,176.546,16.607,152.232
C08029=1096.925,116.681,-62.210,176.544,16.607,152.232
C08030=1096.920,116.432,-62.192,176.541,16.606,152.233
C08031=1096.913,116.183,-62.173,176.538,16.605,152.233
C08032=1096.908,115.933,-62.154,176.536,16.605,152.234
C08033=1096.903,115.685,-62.135,176.533,16.605,152.234
C08034=1096.897,115.435,-62.116,176.530,16.604,152.234
C08035=1096.891,115.186,-62.096,176.527,16.604,152.235
C08036=1096.886,114.937,-62.077,176.525,16.603,152.235
C08037=1096.880,114.688,-62.058,176.522,16.602,152.236
C08038=1096.875,114.438,-62.039,176.519,16.602,152.236
C08039=1096.870,114.189,-62.021,176.516,16.601,152.237
C08040=1096.864,113.940,-62.002,176.514,16.601,152.237
C08041=1096.858,113.690,-61.983,176.511,16.600,152.238
C08042=1096.852,113.441,-61.964,176.509,16.600,152.238
C08043=1096.847,113.192,-61.945,176.505,16.600,152.239
C08044=1096.841,112.943,-61.926,176.503,16.599,152.239
C08045=1096.835,112.693,-61.907,176.500,16.599,152.239
C08046=1096.830,112.445,-61.888,176.497,16.598,152.240
C08047=1096.824,112.170,-61.867,176.494,16.598,152.240
C08048=1096.818,111.895,-61.847,176.492,16.597,152.241
C08049=1096.811,111.620,-61.825,176.489,16.596,152.241
C08050=1096.805,111.345,-61.805,176.486,16.596,152.242
C08051=1096.799,111.096,-61.786,176.483,16.595,152.242
C08052=1096.793,110.847,-61.768,176.481,16.595,152.243
C08053=1096.788,110.597,-61.749,176.478,16.594,152.243
C08054=1096.782,110.348,-61.730,176.475,16.593,152.243
C08055=1096.777,110.099,-61.712,176.472,16.594,152.244
C08056=1096.771,109.850,-61.692,176.469,16.593,152.244
C08057=1096.765,109.600,-61.674,176.467,16.593,152.245
C08058=1096.760,109.351,-61.656,176.464,16.592,152.245
C08059=1096.754,109.102,-61.636,176.461,16.591,152.246
C08060=1096.748,108.853,-61.618,176.459,16.591,152.246
C08061=1096.743,108.604,-61.599,176.456,16.590,152.247
C08062=1096.737,108.354,-61.580,176.454,16.590,152.247
C08063=1096.731,108.105,-61.562,176.451,16.589,152.247
C08064=1096.726,107.856,-61.543,176.448,16.588,152.248
C08065=1096.719,107.607,-61.525,176.445,16.588,152.248
C08066=1096.714,107.358,-61.506,176.442,16.588,152.249
C08067=1096.709,107.108,-61.487,176.440,16.587,152.249
C08068=1096.703,106.859,-61.469,176.437,16.587,152.250
C08069=1096.698,106.609,-61.451,176.435,16.586,152.250
C08070=1096.691,106.360,-61.432,176.432,16.586,152.250
C08071=1096.686,106.111,-61.413,176.429,16.585,152.251
C08072=1096.680,105.862,-61.395,176.427,16.584,152.251
C08073=1096.674,105.612,-61.376,176.424,16.584,152.252
C08074=1096.670,105.363,-61.358,176.422,16.583,152.252
C08075=1096.663,105.114,-61.339,176.419,16.583,152.252
C08076=1096.658,104.865,-61.320,176.416,16.582,152.253
C08077=1096.652,104.615,-61.302,176.413,16.582,152.253
C08078=1096.647,104.367,-61.283,176.410,16.581,152.254
C08079=1096.641,104.117,-61.265,176.409,16.580,152.254
C08080=1096.636,103.868,-61.247,176.406,16.579,152.254
C08081=1096.630,103.618,-61.229,176.403,16.579,152.255
C08082=1096.624,103.370,-61.210,176.400,16.578,152.255
C08083=1096.618,103.120,-61.192,176.397,16.577,152.256
C08084=1096.613,102.871,-61.173,176.395,16.577,152.256
C08085=1096.607,102.621,-61.155,176.392,16.576,152.256
C08086=1096.602,102.373,-61.136,176.390,16.576,152.257
C08087=1096.596,102.123,-61.118,176.387,16.575,152.257
C08088=1096.591,101.874,-61.099,176.385,16.575,152.258
C08089=1096.585,101.624,-61.081,176.382,16.574,152.258
C08090=1096.580,101.375,-61.063,176.379,16.573,152.258
C08091=1096.574,101.126,-61.045,176.377,16.573,152.259
C08092=1096.569,100.877,-61.026,176.374,16.572,152.259
C08093=1096.562,100.628,-61.008,176.372,16.572,152.260
C08094=1096.556,100.378,-60.990,176.369,16.571,152.260
C08095=1096.551,100.128,-60.972,176.367,16.571,152.260
C08096=1096.545,99.879,-60.953,176.364,16.570,152.261
C08097=1096.540,99.630,-60.935,176.361,16.569,152.261
C08098=1096.534,99.381,-60.916,176.359,16.569,152.262
C08099=1096.528,99.132,-60.899,176.356,16.568,152.262
C08100=1096.522,98.882,-60.881,176.354,16.567,152.262
C08101=1096.516,98.634,-60.862,176.351,16.567,152.263
C08102=1096.511,98.384,-60.844,176.349,16.566,152.263
C08103=1096.505,98.135,-60.826,176.346,16.566,152.264
C08104=1096.500,97.885,-60.809,176.343,16.565,152.264
C08105=1096.494,97.636,-60.789,176.341,16.564,152.264
C08106=1096.489,97.387,-60.772,176.338,16.563,152.265
C08107=1096.483,97.137,-60.754,176.336,16.563,152.265
C08108=1096.478,96.889,-60.735,176.333,16.562,152.266
C08109=1096.471,96.639,-60.717,176.330,16.562,152.266
C08110=1096.466,96.390,-60.700,176.328,16.561,152.266
C08111=1096.459,96.115,-60.679,176.325,16.560,152.267
C08112=1096.453,95.841,-60.660,176.323,16.560,152.267
C08113=1096.447,95.565,-60.640,176.320,16.559,152.267
C08114=1096.441,95.291,-60.620,176.317,16.558,152.268
C08115=1096.435,95.041,-60.602,176.314,16.557,152.268
C08116=1096.430,94.792,-60.584,176.311,16.557,152.269
C08117=1096.424,94.543,-60.565,176.309,16.556,152.269
C08118=1096.418,94.294,-60.548,176.307,16.556,152.269
C08119=1096.413,94.045,-60.530,176.304,16.555,152.270
C08120=1096.407,93.795,-60.512,176.302,16.554,152.270
C08121=1096.402,93.546,-60.494,176.299,16.553,152.271
C08122=1096.396,93.296,-60.476,176.297,16.553,152.271
C08123=1096.390,93.047,-60.459,176.294,16.552,152.271
C08124=1096.384,92.798,-60.440,176.292,16.552,152.272
C08125=1096.379,92.548,-60.422,176.289,16.551,152.272
C08126=1096.374,92.299,-60.404,176.286,16.550,152.272
C08127=1096.368,92.050,-60.387,176.284,16.549,152.273
C08128=1096.362,91.801,-60.369,176.281,16.549,152.273
C08129=1096.356,91.551,-60.351,176.279,16.548,152.273
C08130=1096.352,91.302,-60.333,176.276,16.547,152.274
C08131=1096.346,91.052,-60.315,176.274,16.546,152.274
C08132=1096.340,90.803,-60.298,176.271,16.546,152.274
C08133=1096.334,90.554,-60.280,176.269,16.545,152.275
C08134=1096.328,90.305,-60.262,176.266,16.544,152.275
C08135=1096.323,90.056,-60.244,176.264,16.544,152.276
C08136=1096.317,89.806,-60.227,176.261,16.543,152.276
C08137=1096.311,89.557,-60.209,176.259,16.542,152.276
C08138=1096.306,89.308,-60.191,176.256,16.542,152.277
C08139=1096.300,89.058,-60.173,176.253,16.541,152.277
C08140=1096.294,88.809,-60.156,176.251,16.540,152.277
C08141=1096.289,88.560,-60.138,176.248,16.539,152.278
C08142=1096.282,88.310,-60.120,176.246,16.539,152.278
C08143=1096.277,88.061,-60.103,176.243,16.538,152.278
C08144=1096.271,87.812,-60.085,176.241,16.538,152.279
C08145=1096.265,87.562,-60.067,176.239,16.536,152.279
C08146=1096.260,87.313,-60.050,176.236,16.536,152.280
C08147=1096.254,87.064,-60.032,176.233,16.535,152.280
C08148=1096.248,86.814,-60.015,176.232,16.535,152.280
C08149=1096.243,86.565,-59.997,176.229,16.534,152.281
C08150=1096.237,86.316,-59.980,176.227,16.533,152.281
C08151=1096.231,86.066,-59.962,176.224,16.532,152.281
C08152=1096.226,85.817,-59.944,176.222,16.532,152.282
C08153=1096.220,85.568,-59.927,176.219,16.531,152.282
C08154=1096.215,85.319,-59.909,176.217,16.530,152.282
C08155=1096.209,85.069,-59.892,176.214,16.529,152.283
C08156=1096.203,84.820,-59.874,176.212,16.529,152.283
C08157=1096.198,84.570,-59.857,176.209,16.528,152.283
C08158=1096.192,84.321,-59.839,176.207,16.527,152.284
C08159=1096.185,84.072,-59.822,176.204,16.526,152.284
C08160=1096.180,83.822,-59.805,176.202,16.525,152.284
C08161=1096.175,83.573,-59.788,176.199,16.525,152.285
C08162=1096.169,83.324,-59.770,176.197,16.524,152.285
C08163=1096.163,83.075,-59.752,176.194,16.523,152.285
C08164=1096.158,82.825,-59.734,176.192,16.522,152.286
C08165=1096.152,82.576,-59.718,176.190,16.522,152.286
C08166=1096.147,82.327,-59.700,176.187,16.521,152.286
C08167=1096.141,82.077,-59.682,176.185,16.520,152.287
C08168=1096.136,81.827,-59.665,176.182,16.519,152.287
C08169=1096.130,81.578,-59.648,176.180,16.519,152.287
C08170=1096.124,81.329,-59.630,176.177,16.518,152.288
C08171=1096.119,81.080,-59.614,176.175,16.517,152.288
C08172=1096.112,80.830,-59.596,176.173,16.516,152.288
C08173=1096.107,80.581,-59.578,176.170,16.516,152.289
C08174=1096.102,80.332,-59.562,176.168,16.514,152.289
C08175=1096.096,80.057,-59.542,176.165,16.514,152.289
C08176=1096.089,79.783,-59.523,176.163,16.513,152.290
C08177=1096.084,79.508,-59.504,176.160,16.512,152.290
C08178=1096.077,79.233,-59.485,176.157,16.511,152.290
C08179=1096.071,78.984,-59.467,176.155,16.510,152.290
C08180=1096.066,78.734,-59.451,176.152,16.509,152.291
C08181=1096.060,78.485,-59.434,176.150,16.509,152.291
C08182=1096.055,78.236,-59.417,176.147,16.508,152.292
C08183=1096.048,77.986,-59.399,176.145,16.507,152.292
C08184=1096.043,77.737,-59.381,176.143,16.506,152.292
C08185=1096.037,77.488,-59.365,176.141,16.506,152.293
C08186=1096.031,77.239,-59.347,176.138,16.504,152.293
C08187=1096.026,76.989,-59.331,176.136,16.504,152.293
C08188=1096.020,76.740,-59.314,176.133,16.503,152.293
C08189=1096.014,76.490,-59.296,176.131,16.502,152.294
C08190=1096.009,76.241,-59.279,176.128,16.501,152.294
C08191=1096.003,75.991,-59.262,176.126,16.501,152.294
C08192=1095.997,75.742,-59.245,176.124,16.499,152.295
C08193=1095.992,75.493,-59.228,176.122,16.499,152.295
C08194=1095.986,75.244,-59.211,176.119,16.498,152.295
C08195=1095.980,74.994,-59.194,176.117,16.497,152.296
C08196=1095.974,74.745,-59.176,176.114,16.496,152.296
C08197=1095.968,74.495,-59.160,176.112,16.495,152.296
C08198=1095.963,74.246,-59.143,176.109,16.495,152.297
C08199=1095.958,73.997,-59.126,176.107,16.494,152.297
C08200=1095.952,73.747,-59.109,176.105,16.493,152.297
C08201=1095.946,73.498,-59.092,176.103,16.492,152.297
C08202=1095.941,73.248,-59.075,176.100,16.491,152.298
C08203=1095.935,73.000,-59.058,176.098,16.490,152.298
C08204=1095.930,72.750,-59.041,176.095,16.489,152.298
C08205=1095.924,72.500,-59.024,176.093,16.489,152.299
C08206=1095.918,72.252,-59.007,176.091,16.488,152.299
C08207=1095.912,72.001,-58.990,176.088,16.487,152.299
C08208=1095.906,71.752,-58.974,176.087,16.486,152.299
C08209=1095.901,71.503,-58.956,176.084,16.485,152.300
C08210=1095.896,71.253,-58.940,176.082,16.484,152.300
C08211=1095.890,71.004,-58.923,176.079,16.484,152.300
C08212=1095.884,70.755,-58.906,176.077,16.483,152.301
C08213=1095.878,70.506,-58.889,176.074,16.482,152.301
C08214=1095.873,70.256,-58.873,176.072,16.481,152.301
C08215=1095.867,70.007,-58.856,176.070,16.480,152.301
C08216=1095.861,69.758,-58.839,176.068,16.479,152.302
C08217=1095.856,69.508,-58.822,176.065,16.478,152.302
C08218=1095.850,69.259,-58.806,176.063,16.478,152.302
C08219=1095.844,69.010,-58.789,176.060,16.476,152.303
C08220=1095.839,68.760,-58.772,176.058,16.476,152.303
C08221=1095.833,68.511,-58.756,176.056,16.474,152.303
C08222=1095.828,68.261,-58.739,176.054,16.474,152.303
C08223=1095.821,68.012,-58.722,176.051,16.473,152.304
C08224=1095.816,67.763,-58.705,176.049,16.472,152.304
C08225=1095.810,67.513,-58.689,176.047,16.472,152.304
C08226=1095.805,67.264,-58.672,176.044,16.470,152.305
C08227=1095.799,67.014,-58.656,176.042,16.470,152.305
C08228=1095.794,66.765,-58.638,176.040,16.468,152.305
C08229=1095.788,66.516,-58.622,176.038,16.468,152.305
C08230=1095.782,66.267,-58.605,176.035,16.467,152.306
C08231=1095.776,66.017,-58.589,176.033,16.466,152.306
C08232=1095.770,65.768,-58.572,176.030,16.465,152.306
C08233=1095.765,65.518,-58.555,176.028,16.464,152.307
C08234=1095.759,65.269,-58.539,176.026,16.463,152.307
C08235=1095.753,65.020,-58.522,176.024,16.462,152.307
C08236=1095.748,64.770,-58.505,176.021,16.461,152.307
C08237=1095.742,64.521,-58.489,176.019,16.460,152.308
C08238=1095.737,64.271,-58.472,176.017,16.460,152.308
C08239=1095.730,63.997,-58.454,176.014,16.459,152.308
C08240=1095.724,63.722,-58.436,176.012,16.458,152.309
C08241=1095.717,63.447,-58.418,176.009,16.456,152.309
C08242=1095.710,63.172,-58.400,176.007,16.456,152.309
C08243=1095.705,62.922,-58.383,176.004,16.454,152.310
C08244=1095.699,62.673,-58.367,176.003,16.454,152.310
C08245=1095.693,62.424,-58.351,176.000,16.453,152.310
C08246=1095.687,62.174,-58.334,175.998,16.452,152.310
C08247=1095.681,61.925,-58.318,175.996,16.452,152.311
C08248=1095.676,61.675,-58.302,175.993,16.450,152.311
C08249=1095.670,61.426,-58.285,175.991,16.450,152.311
C08250=1095.664,61.176,-58.268,175.988,16.448,152.311
C08251=1095.659,60.928,-58.253,175.987,16.448,152.312
C08252=1095.653,60.678,-58.236,175.984,16.446,152.312
C08253=1095.647,60.429,-58.220,175.982,16.446,152.312
C08254=1095.641,60.179,-58.204,175.979,16.444,152.313
C08255=1095.636,59.930,-58.187,175.977,16.444,152.313
C08256=1095.630,59.680,-58.171,175.976,16.443,152.313
C08257=1095.624,59.431,-58.154,175.973,16.442,152.313
C08258=1095.618,59.182,-58.138,175.971,16.441,152.314
C08259=1095.612,58.932,-58.122,175.968,16.440,152.314
C08260=1095.606,58.683,-58.106,175.966,16.439,152.314
C08261=1095.601,58.433,-58.089,175.964,16.438,152.314
C08262=1095.595,58.184,-58.073,175.962,16.437,152.315
C08263=1095.589,57.934,-58.057,175.960,16.437,152.315
C08264=1095.583,57.685,-58.041,175.957,16.435,152.315
C08265=1095.577,57.435,-58.025,175.955,16.435,152.315
C08266=1095.572,57.187,-58.009,175.953,16.433,152.316
C08267=1095.566,56.937,-57.992,175.951,16.433,152.316
C08268=1095.561,56.688,-57.976,175.948,16.431,152.316
C08269=1095.555,56.438,-57.959,175.946,16.431,152.316
C08270=1095.549,56.188,-57.944,175.944,16.430,152.317
C08271=1095.543,55.939,-57.927,175.941,16.429,152.317
C08272=1095.537,55.690,-57.911,175.940,16.428,152.317
C08273=1095.531,55.440,-57.895,175.937,16.427,152.318
C08274=1095.526,55.192,-57.879,175.935,16.426,152.318
C08275=1095.520,54.942,-57.864,175.933,16.424,152.318
C08276=1095.515,54.692,-57.847,175.931,16.424,152.318
C08277=1095.509,54.443,-57.830,175.929,16.423,152.318
C08278=1095.503,54.193,-57.814,175.926,16.422,152.319
C08279=1095.498,53.943,-57.799,175.924,16.421,152.319
C08280=1095.492,53.695,-57.783,175.922,16.420,152.319
C08281=1095.486,53.445,-57.766,175.920,16.419,152.319
C08282=1095.481,53.195,-57.751,175.917,16.418,152.320
C08283=1095.475,52.946,-57.735,175.915,16.417,152.320
C08284=1095.469,52.697,-57.718,175.913,16.416,152.320
C08285=1095.464,52.448,-57.703,175.911,16.415,152.320
C08286=1095.458,52.198,-57.687,175.909,16.414,152.321
C08287=1095.452,51.949,-57.671,175.906,16.413,152.321
C08288=1095.446,51.699,-57.654,175.904,16.412,152.321
C08289=1095.440,51.450,-57.639,175.903,16.411,152.321
C08290=1095.436,51.201,-57.622,175.900,16.410,152.322
C08291=1095.430,50.951,-57.607,175.898,16.409,152.322
C08292=1095.424,50.701,-57.591,175.895,16.408,152.322
C08293=1095.418,50.452,-57.574,175.894,16.407,152.322
C08294=1095.413,50.203,-57.559,175.891,16.405,152.322
C08295=1095.407,49.953,-57.543,175.889,16.405,152.323
C08296=1095.402,49.703,-57.527,175.887,16.404,152.323
C08297=1095.396,49.454,-57.511,175.885,16.403,152.323
C08298=1095.390,49.205,-57.495,175.883,16.402,152.323
C08299=1095.385,48.955,-57.480,175.880,16.400,152.324
C08300=1095.379,48.706,-57.463,175.878,16.400,152.324
C08301=1095.373,48.456,-57.448,175.877,16.399,152.324
C08302=1095.368,48.207,-57.432,175.874,16.397,152.324
C08303=1095.361,47.933,-57.415,175.872,16.397,152.324
C08304=1095.355,47.657,-57.398,175.870,16.395,152.325
C08305=1095.349,47.382,-57.380,175.867,16.394,152.325
C08306=1095.342,47.107,-57.363,175.865,16.393,152.325
C08307=1095.337,46.858,-57.347,175.863,16.392,152.325
C08308=1095.331,46.608,-57.331,175.861,16.391,152.326
C08309=1095.326,46.358,-57.316,175.858,16.390,152.326
C08310=1095.320,46.110,-57.300,175.856,16.389,152.326
C08311=1095.315,45.860,-57.284,175.854,16.388,152.326
C08312=1095.309,45.610,-57.268,175.852,16.387,152.327
C08313=1095.304,45.361,-57.253,175.850,16.385,152.327
C08314=1095.298,45.112,-57.236,175.847,16.384,152.327
C08315=1095.292,44.862,-57.221,175.846,16.384,152.327
C08316=1095.287,44.613,-57.205,175.844,16.382,152.327
C08317=1095.281,44.363,-57.189,175.841,16.381,152.328
C08318=1095.275,44.113,-57.174,175.839,16.380,152.328
C08319=1095.270,43.865,-57.158,175.837,16.379,152.328
C08320=1095.264,43.615,-57.143,175.835,16.378,152.328
C08321=1095.258,43.366,-57.127,175.833,16.377,152.328
C08322=1095.253,43.116,-57.112,175.831,16.376,152.329
C08323=1095.247,42.866,-57.096,175.829,16.375,152.329
C08324=1095.241,42.617,-57.080,175.826,16.374,152.329
C08325=1095.235,42.368,-57.065,175.825,16.372,152.329
C08326=1095.230,42.118,-57.050,175.823,16.372,152.329
C08327=1095.224,41.869,-57.034,175.820,16.371,152.330
C08328=1095.219,41.619,-57.018,175.818,16.369,152.330
C08329=1095.213,41.369,-57.003,175.817,16.369,152.330
C08330=1095.206,41.120,-56.987,175.814,16.367,152.330
C08331=1095.201,40.871,-56.972,175.812,16.366,152.330
C08332=1095.196,40.621,-56.956,175.810,16.365,152.331
C08333=1095.191,40.372,-56.941,175.808,16.364,152.331
C08334=1095.184,40.123,-56.926,175.806,16.363,152.331
C08335=1095.178,39.873,-56.910,175.803,16.362,152.331
C08336=1095.173,39.624,-56.895,175.801,16.361,152.332
C08337=1095.167,39.374,-56.879,175.800,16.360,152.332
C08338=1095.161,39.125,-56.864,175.797,16.359,152.332
C08339=1095.156,38.875,-56.848,175.796,16.358,152.332
C08340=1095.150,38.625,-56.833,175.793,16.356,152.332
C08341=1095.145,38.376,-56.818,175.791,16.356,152.333
C08342=1095.138,38.127,-56.802,175.789,16.355,152.333
C08343=1095.133,37.878,-56.787,175.787,16.353,152.333
C08344=1095.128,37.628,-56.771,175.785,16.352,152.333
C08345=1095.121,37.378,-56.756,175.783,16.351,152.333
C08346=1095.116,37.129,-56.741,175.780,16.350,152.334
C08347=1095.110,36.880,-56.726,175.779,16.349,152.334
C08348=1095.104,36.630,-56.710,175.776,16.348,152.334
C08349=1095.099,36.381,-56.695,175.774,16.347,152.334
C08350=1095.093,36.131,-56.680,175.773,16.346,152.334
C08351=1095.087,35.882,-56.665,175.770,16.345,152.335
C08352=1095.081,35.632,-56.650,175.768,16.344,152.335
C08353=1095.075,35.382,-56.634,175.766,16.343,152.335
C08354=1095.069,35.134,-56.619,175.764,16.342,152.335
C08355=1095.064,34.884,-56.603,175.762,16.340,152.335
C08356=1095.058,34.635,-56.589,175.760,16.340,152.336
C08357=1095.052,34.385,-56.573,175.758,16.338,152.336
C08358=1095.047,34.136,-56.558,175.756,16.337,152.336
C08359=1095.041,33.886,-56.543,175.754,16.337,152.336
C08360=1095.035,33.636,-56.528,175.752,16.335,152.336
C08361=1095.029,33.387,-56.513,175.750,16.334,152.337
C08362=1095.024,33.137,-56.498,175.748,16.333,152.337
C08363=1095.018,32.888,-56.483,175.746,16.332,152.337
C08364=1095.012,32.638,-56.467,175.744,16.331,152.337
C08365=1095.007,32.389,-56.453,175.741,16.329,152.337
C08366=1095.001,32.139,-56.437,175.740,16.328,152.338
C08367=1094.995,31.865,-56.420,175.738,16.328,152.338
C08368=1094.988,31.590,-56.404,175.735,16.326,152.338
C08369=1094.982,31.314,-56.387,175.733,16.325,152.338
C08370=1094.976,31.040,-56.371,175.731,16.324,152.338
C08371=1094.970,30.790,-56.356,175.728,16.322,152.339
C08372=1094.964,30.541,-56.341,175.726,16.322,152.339
C08373=1094.959,30.291,-56.326,175.725,16.320,152.339
C08374=1094.953,30.042,-56.311,175.722,16.319,152.339
C08375=1094.947,29.792,-56.296,175.721,16.318,152.339
C08376=1094.942,29.543,-56.281,175.719,16.317,152.340
C08377=1094.935,29.293,-56.266,175.716,16.316,152.340
C08378=1094.930,29.044,-56.251,175.714,16.315,152.340
C08379=1094.924,28.795,-56.236,175.713,16.314,152.340
C08380=1094.919,28.545,-56.221,175.710,16.312,152.340
C08381=1094.913,28.296,-56.206,175.708,16.311,152.340
C08382=1094.907,28.046,-56.190,175.707,16.311,152.341
C08383=1094.902,27.796,-56.177,175.704,16.309,152.341
C08384=1094.895,27.547,-56.162,175.702,16.308,152.341
C08385=1094.890,27.297,-56.146,175.701,16.307,152.341
C08386=1094.884,27.048,-56.132,175.698,16.306,152.341
C08387=1094.878,26.799,-56.117,175.696,16.305,152.342
C08388=1094.873,26.549,-56.101,175.695,16.303,152.342
C08389=1094.867,26.300,-56.087,175.692,16.302,152.342
C08390=1094.861,26.050,-56.073,175.690,16.301,152.342
C08391=1094.856,25.800,-56.057,175.689,16.300,152.342
C08392=1094.849,25.551,-56.042,175.686,16.299,152.342
C08393=1094.843,25.302,-56.028,175.684,16.298,152.343
C08394=1094.838,25.052,-56.012,175.683,16.297,152.343
C08395=1094.832,24.802,-55.998,175.681,16.296,152.343
C08396=1094.826,24.553,-55.984,175.678,16.294,152.343
C08397=1094.820,24.304,-55.969,175.676,16.294,152.343
C08398=1094.815,24.054,-55.954,175.675,16.293,152.343
C08399=1094.809,23.804,-55.940,175.672,16.291,152.344
C08400=1094.803,23.555,-55.925,175.671,16.290,152.344
C08401=1094.798,23.305,-55.909,175.669,16.289,152.344
C08402=1094.792,23.056,-55.895,175.666,16.288,152.344
C08403=1094.786,22.806,-55.881,175.665,16.287,152.344
C08404=1094.780,22.557,-55.866,175.663,16.286,152.345
C08405=1094.775,22.308,-55.851,175.660,16.284,152.345
C08406=1094.769,22.057,-55.837,175.658,16.283,152.345
C08407=1094.763,21.808,-55.822,175.657,16.282,152.345
C08408=1094.757,21.560,-55.807,175.654,16.281,152.345
C08409=1094.752,21.309,-55.793,175.653,16.280,152.345
C08410=1094.746,21.060,-55.778,175.651,16.279,152.346
C08411=1094.740,20.810,-55.763,175.649,16.278,152.346
C08412=1094.734,20.561,-55.749,175.647,16.276,152.346
C08413=1094.729,20.311,-55.734,175.645,16.275,152.346
C08414=1094.723,20.062,-55.719,175.643,16.274,152.346
C08415=1094.717,19.812,-55.705,175.641,16.273,152.346
C08416=1094.711,19.563,-55.690,175.639,16.272,152.346
C08417=1094.705,19.314,-55.676,175.637,16.271,152.347
C08418=1094.701,19.064,-55.661,175.635,16.269,152.347
C08419=1094.694,18.814,-55.646,175.633,16.268,152.347
C08420=1094.689,18.565,-55.632,175.631,16.267,152.347
C08421=1094.683,18.316,-55.618,175.630,16.266,152.347
C08422=1094.677,18.065,-55.604,175.627,16.265,152.348
C08423=1094.671,17.816,-55.589,175.625,16.264,152.348
C08424=1094.665,17.567,-55.575,175.624,16.263,152.348
C08425=1094.659,17.317,-55.560,175.621,16.261,152.348
C08426=1094.654,17.068,-55.545,175.620,16.260,152.348
C08427=1094.649,16.818,-55.531,175.618,16.260,152.348
C08428=1094.642,16.569,-55.516,175.616,16.258,152.349
C08429=1094.637,16.319,-55.502,175.614,16.257,152.349
C08430=1094.631,16.070,-55.488,175.612,16.256,152.349
C08431=1094.624,15.796,-55.472,175.609,16.254,152.349
C08432=1094.618,15.523,-55.456,175.608,16.253,152.349
C08433=1094.612,15.249,-55.441,175.605,16.252,152.349
C08434=1094.606,14.976,-55.425,175.603,16.251,152.350
C08435=1094.600,14.725,-55.410,175.602,16.250,152.350
C08436=1094.595,14.476,-55.396,175.599,16.248,152.350
C08437=1094.589,14.227,-55.382,175.598,16.247,152.350
C08438=1094.583,13.977,-55.367,175.596,16.246,152.350
C08439=1094.577,13.727,-55.353,175.594,16.245,152.350
C08440=1094.571,13.479,-55.339,175.592,16.243,152.351
C08441=1094.565,13.229,-55.325,175.590,16.243,152.351
C08442=1094.559,12.980,-55.310,175.588,16.242,152.351
C08443=1094.553,12.730,-55.296,175.586,16.240,152.351
C08444=1094.547,12.480,-55.282,175.584,16.239,152.351
C08445=1094.541,12.231,-55.268,175.582,16.238,152.351
C08446=1094.536,11.981,-55.254,175.580,16.237,152.352
C08447=1094.530,11.731,-55.240,175.578,16.236,152.352
C08448=1094.524,11.482,-55.225,175.576,16.235,152.352
C08449=1094.519,11.232,-55.211,175.575,16.234,152.352
C08450=1094.512,10.983,-55.196,175.573,16.233,152.352
C08451=1094.507,10.733,-55.182,175.571,16.231,152.352
C08452=1094.501,10.484,-55.169,175.569,16.230,152.353
C08453=1094.495,10.235,-55.154,175.567,16.229,152.353
C08454=1094.489,9.985,-55.140,175.565,16.228,152.353
C08455=1094.483,9.735,-55.126,175.563,16.227,152.353
C08456=1094.477,9.486,-55.112,175.561,16.226,152.353
C08457=1094.471,9.236,-55.098,175.560,16.224,152.353
C08458=1094.466,8.986,-55.084,175.558,16.224,152.354
C08459=1094.460,8.737,-55.070,175.555,16.222,152.354
C08460=1094.454,8.488,-55.056,175.554,16.221,152.354
C08461=1094.448,8.238,-55.042,175.552,16.220,152.354
C08462=1094.442,7.988,-55.028,175.549,16.218,152.354
C08463=1094.437,7.739,-55.014,175.548,16.217,152.354
C08464=1094.431,7.490,-54.999,175.546,16.217,152.354
C08465=1094.425,7.239,-54.985,175.544,16.215,152.355
C08466=1094.420,6.990,-54.971,175.542,16.214,152.355
C08467=1094.413,6.741,-54.958,175.540,16.213,152.355
C08468=1094.408,6.492,-54.943,175.538,16.212,152.355
C08469=1094.402,6.242,-54.930,175.537,16.211,152.355
C08470=1094.396,5.992,-54.915,175.534,16.209,152.355
C08471=1094.391,5.742,-54.901,175.532,16.208,152.356
C08472=1094.385,5.493,-54.888,175.531,16.207,152.356
C08473=1094.379,5.244,-54.874,175.529,16.206,152.356
C08474=1094.373,4.994,-54.860,175.527,16.204,152.356
C08475=1094.367,4.744,-54.845,175.525,16.204,152.356
C08476=1094.362,4.495,-54.832,175.523,16.202,152.356
C08477=1094.356,4.245,-54.818,175.522,16.201,152.356
C08478=1094.350,3.996,-54.804,175.520,16.200,152.356
C08479=1094.344,3.746,-54.791,175.517,16.199,152.357
C08480=1094.339,3.497,-54.777,175.516,16.198,152.357
C08481=1094.332,3.247,-54.762,175.514,16.197,152.357
C08482=1094.327,2.997,-54.748,175.513,16.195,152.357
C08483=1094.321,2.748,-54.735,175.510,16.194,152.357
C08484=1094.315,2.498,-54.721,175.508,16.193,152.357
C08485=1094.310,2.249,-54.707,175.507,16.192,152.357
C08486=1094.304,1.999,-54.693,175.505,16.191,152.358
C08487=1094.299,1.750,-54.679,175.503,16.189,152.358
C08488=1094.292,1.500,-54.666,175.501,16.188,152.358
C08489=1094.287,1.250,-54.652,175.499,16.187,152.358
C08490=1094.281,1.001,-54.638,175.498,16.186,152.358
C08491=1094.276,0.751,-54.624,175.495,16.184,152.358
C08492=1094.269,0.502,-54.611,175.494,16.183,152.358
C08493=1094.264,0.252,-54.597,175.492,16.182,152.359
C08494=1094.258,0.003,-54.583,175.490,16.181,152.359
C08495=1094.252,-0.269,-54.568,175.488,16.179,152.359
C08496=1094.246,-0.540,-54.553,175.486,16.178,152.359
C08497=1094.239,-0.812,-54.538,175.483,16.177,152.359
C08498=1094.233,-1.083,-54.523,175.482,16.176,152.359
C08499=1094.228,-1.333,-54.509,175.480,16.175,152.360
C08500=1094.222,-1.582,-54.496,175.479,16.174,152.360
C08501=1094.216,-1.832,-54.482,175.476,16.172,152.360
C08502=1094.211,-2.081,-54.468,175.475,16.171,152.360
C08503=1094.205,-2.331,-54.454,175.473,16.170,152.360
C08504=1094.198,-2.581,-54.441,175.471,16.169,152.360
C08505=1094.193,-2.831,-54.427,175.469,16.167,152.360
C08506=1094.188,-3.080,-54.413,175.467,16.166,152.360
C08507=1094.182,-3.330,-54.400,175.466,16.165,152.361
C08508=1094.176,-3.580,-54.387,175.464,16.164,152.361
C08509=1094.170,-3.829,-54.373,175.462,16.163,152.361
C08510=1094.164,-4.078,-54.359,175.460,16.161,152.361
C08511=1094.159,-4.328,-54.346,175.458,16.160,152.361
C08512=1094.153,-4.577,-54.332,175.456,16.159,152.361
C08513=1094.147,-4.827,-54.318,175.455,16.158,152.361
C08514=1094.141,-5.076,-54.305,175.453,16.157,152.362
C08515=1094.135,-5.326,-54.291,175.451,16.155,152.362
C08516=1094.129,-5.576,-54.278,175.449,16.154,152.362
C08517=1094.124,-5.826,-54.265,175.447,16.153,152.362
C08518=1094.117,-6.075,-54.251,175.445,16.152,152.362
C08519=1094.112,-6.325,-54.237,175.444,16.151,152.362
C08520=1094.106,-6.574,-54.224,175.441,16.149,152.362
C08521=1094.100,-6.823,-54.211,175.440,16.149,152.363
C08522=1094.094,-7.073,-54.198,175.438,16.148,152.363
C08523=1094.088,-7.323,-54.184,175.436,16.146,152.363
C08524=1094.083,-7.572,-54.171,175.435,16.145,152.363
C08525=1094.076,-7.822,-54.157,175.432,16.144,152.363
C08526=1094.071,-8.072,-54.144,175.430,16.143,152.363
C08527=1094.065,-8.321,-54.131,175.429,16.142,152.363
C08528=1094.060,-8.571,-54.117,175.427,16.141,152.364
C08529=1094.053,-8.820,-54.104,175.426,16.139,152.364
C08530=1094.048,-9.069,-54.090,175.423,16.138,152.364
C08531=1094.042,-9.319,-54.077,175.421,16.137,152.364
C08532=1094.037,-9.569,-54.064,175.420,16.136,152.364
C08533=1094.030,-9.818,-54.050,175.418,16.135,152.364
C08534=1094.024,-10.068,-54.038,175.417,16.133,152.364
C08535=1094.019,-10.318,-54.024,175.414,16.132,152.364
C08536=1094.013,-10.567,-54.011,175.412,16.131,152.365
C08537=1094.007,-10.816,-53.997,175.411,16.130,152.365
C08538=1094.001,-11.066,-53.984,175.409,16.129,152.365
C08539=1093.996,-11.316,-53.970,175.407,16.128,152.365
C08540=1093.990,-11.565,-53.957,175.406,16.126,152.365
C08541=1093.984,-11.815,-53.944,175.403,16.125,152.365
C08542=1093.978,-12.065,-53.931,175.402,16.124,152.366
C08543=1093.972,-12.314,-53.918,175.400,16.123,152.366
C08544=1093.967,-12.564,-53.904,175.398,16.122,152.366
C08545=1093.961,-12.813,-53.891,175.397,16.121,152.366
C08546=1093.955,-13.063,-53.878,175.394,16.119,152.366
C08547=1093.949,-13.313,-53.864,175.393,16.118,152.366
C08548=1093.943,-13.562,-53.851,175.391,16.117,152.366
C08549=1093.938,-13.812,-53.838,175.389,16.116,152.366
C08550=1093.932,-14.061,-53.825,175.388,16.115,152.366
C08551=1093.926,-14.311,-53.812,175.386,16.114,152.367
C08552=1093.920,-14.561,-53.798,175.384,16.112,152.367
C08553=1093.914,-14.810,-53.785,175.382,16.111,152.367
C08554=1093.908,-15.060,-53.773,175.380,16.109,152.367
C08555=1093.903,-15.309,-53.759,175.379,16.109,152.367
C08556=1093.897,-15.559,-53.747,175.377,16.108,152.367
C08557=1093.891,-15.808,-53.733,175.375,16.106,152.367
C08558=1093.885,-16.058,-53.721,175.373,16.105,152.368
C08559=1093.878,-16.328,-53.706,175.371,16.104,152.368
C08560=1093.872,-16.598,-53.692,175.369,16.103,152.368
C08561=1093.866,-16.868,-53.678,175.367,16.101,152.368
C08562=1093.860,-17.138,-53.664,175.365,16.100,152.368
C08563=1093.854,-17.388,-53.651,175.364,16.099,152.368
C08564=1093.847,-17.637,-53.638,175.362,16.098,152.368
C08565=1093.842,-17.887,-53.625,175.360,16.097,152.369
C08566=1093.836,-18.137,-53.611,175.359,16.096,152.369
C08567=1093.830,-18.387,-53.599,175.356,16.094,152.369
C08568=1093.825,-18.635,-53.586,175.355,16.093,152.369
C08569=1093.819,-18.885,-53.573,175.353,16.092,152.369
C08570=1093.813,-19.135,-53.560,175.351,16.091,152.369
C08571=1093.807,-19.384,-53.547,175.350,16.090,152.369
C08572=1093.801,-19.634,-53.534,175.348,16.089,152.369
C08573=1093.795,-19.884,-53.521,175.346,16.087,152.370
C08574=1093.789,-20.133,-53.508,175.344,16.086,152.370
C08575=1093.784,-20.383,-53.495,175.342,16.085,152.370
C08576=1093.778,-20.633,-53.482,175.341,16.084,152.370
C08577=1093.772,-20.882,-53.469,175.339,16.083,152.370
C08578=1093.766,-21.131,-53.457,175.337,16.082,152.370
C08579=1093.760,-21.381,-53.443,175.336,16.081,152.370
C08580=1093.754,-21.630,-53.431,175.333,16.079,152.371
C08581=1093.748,-21.880,-53.418,175.331,16.078,152.371
C08582=1093.743,-22.130,-53.404,175.330,16.077,152.371
C08583=1093.737,-22.380,-53.392,175.328,16.076,152.371
C08584=1093.731,-22.630,-53.379,175.327,16.075,152.371
C08585=1093.725,-22.878,-53.366,175.325,16.074,152.371
C08586=1093.719,-23.128,-53.354,175.323,16.072,152.371
C08587=1093.714,-23.378,-53.341,175.322,16.072,152.372
C08588=1093.707,-23.627,-53.328,175.319,16.070,152.372
C08589=1093.702,-23.878,-53.315,175.318,16.069,152.372
C08590=1093.696,-24.127,-53.302,175.316,16.068,152.372
C08591=1093.691,-24.376,-53.289,175.314,16.067,152.372
C08592=1093.685,-24.626,-53.277,175.313,16.065,152.372
C08593=1093.679,-24.876,-53.264,175.311,16.064,152.372
C08594=1093.673,-25.126,-53.252,175.309,16.064,152.372
C08595=1093.667,-25.375,-53.239,175.308,16.062,152.373
C08596=1093.661,-25.624,-53.226,175.305,16.061,152.373
C08597=1093.656,-25.874,-53.214,175.304,16.060,152.373
C08598=1093.650,-26.124,-53.201,175.302,16.058,152.373
C08599=1093.644,-26.373,-53.187,175.300,16.057,152.373
C08600=1093.638,-26.623,-53.175,175.299,16.056,152.373
C08601=1093.633,-26.872,-53.163,175.297,16.055,152.373
C08602=1093.627,-27.122,-53.150,175.295,16.054,152.373
C08603=1093.621,-27.372,-53.137,175.294,16.053,152.374
C08604=1093.615,-27.621,-53.124,175.291,16.051,152.374
C08605=1093.608,-27.871,-53.112,175.290,16.050,152.374
C08606=1093.603,-28.120,-53.100,175.288,16.050,152.374
C08607=1093.597,-28.370,-53.088,175.286,16.048,152.374
C08608=1093.591,-28.619,-53.074,175.285,16.047,152.374
C08609=1093.585,-28.869,-53.062,175.283,16.046,152.374
C08610=1093.579,-29.119,-53.049,175.281,16.045,152.374
C08611=1093.573,-29.369,-53.037,175.280,16.044,152.375
C08612=1093.568,-29.618,-53.024,175.278,16.043,152.375
C08613=1093.562,-29.868,-53.012,175.276,16.042,152.375
C08614=1093.556,-30.117,-52.999,175.274,16.040,152.375
C08615=1093.550,-30.367,-52.986,175.272,16.039,152.375
C08616=1093.544,-30.616,-52.974,175.271,16.038,152.375
C08617=1093.538,-30.866,-52.962,175.269,16.037,152.376
C08618=1093.532,-31.116,-52.949,175.267,16.036,152.376
C08619=1093.526,-31.366,-52.937,175.266,16.035,152.376
C08620=1093.520,-31.616,-52.924,175.264,16.034,152.376
C08621=1093.515,-31.865,-52.912,175.262,16.033,152.376
C08622=1093.509,-32.115,-52.900,175.261,16.032,152.376
C08623=1093.502,-32.383,-52.886,175.258,16.030,152.376
C08624=1093.495,-32.653,-52.872,175.257,16.029,152.376
C08625=1093.490,-32.922,-52.859,175.255,16.028,152.377
C08626=1093.483,-33.191,-52.846,175.253,16.027,152.377
C08627=1093.478,-33.441,-52.833,175.251,16.026,152.377
C08628=1093.472,-33.691,-52.821,175.249,16.024,152.377
C08629=1093.466,-33.940,-52.809,175.247,16.023,152.377
C08630=1093.460,-34.189,-52.796,175.246,16.022,152.377
C08631=1093.454,-34.439,-52.784,175.244,16.021,152.377
C08632=1093.448,-34.689,-52.772,175.243,16.020,152.377
C08633=1093.443,-34.938,-52.759,175.241,16.019,152.378
C08634=1093.437,-35.188,-52.747,175.239,16.018,152.378
C08635=1093.431,-35.438,-52.734,175.238,16.017,152.378
C08636=1093.425,-35.687,-52.722,175.236,16.015,152.378
C08637=1093.419,-35.937,-52.710,175.234,16.014,152.378
C08638=1093.413,-36.187,-52.697,175.233,16.013,152.378
C08639=1093.408,-36.436,-52.685,175.231,16.013,152.378
C08640=1093.402,-36.686,-52.673,175.229,16.011,152.379
C08641=1093.395,-36.935,-52.661,175.227,16.010,152.379
C08642=1093.390,-37.185,-52.648,175.225,16.008,152.379
C08643=1093.384,-37.435,-52.636,175.224,16.007,152.379
C08644=1093.378,-37.684,-52.623,175.222,16.006,152.379
C08645=1093.373,-37.934,-52.611,175.220,16.005,152.379
C08646=1093.367,-38.183,-52.599,175.219,16.004,152.379
C08647=1093.360,-38.433,-52.587,175.217,16.003,152.379
C08648=1093.355,-38.683,-52.575,175.215,16.002,152.380
C08649=1093.349,-38.933,-52.563,175.214,16.001,152.380
C08650=1093.342,-39.182,-52.551,175.212,16.000,152.380
C08651=1093.337,-39.432,-52.538,175.210,15.999,152.380
C08652=1093.331,-39.681,-52.526,175.209,15.998,152.380
C08653=1093.325,-39.931,-52.514,175.207,15.997,152.380
C08654=1093.319,-40.180,-52.502,175.205,15.996,152.380
C08655=1093.313,-40.430,-52.489,175.204,15.995,152.381
C08656=1093.307,-40.680,-52.478,175.202,15.994,152.381
C08657=1093.302,-40.929,-52.466,175.200,15.992,152.381
C08658=1093.296,-41.179,-52.453,175.198,15.991,152.381
C08659=1093.289,-41.429,-52.441,175.196,15.990,152.381
C08660=1093.284,-41.678,-52.429,175.194,15.989,152.381
C08661=1093.277,-41.928,-52.417,175.193,15.988,152.381
C08662=1093.272,-42.178,-52.405,175.191,15.987,152.382
C08663=1093.266,-42.427,-52.393,175.190,15.986,152.382
C08664=1093.260,-42.677,-52.381,175.188,15.985,152.382
C08665=1093.254,-42.927,-52.369,175.186,15.984,152.382
C08666=1093.248,-43.176,-52.356,175.185,15.983,152.382
C08667=1093.242,-43.426,-52.345,175.183,15.981,152.382
C08668=1093.236,-43.676,-52.333,175.181,15.980,152.382
C08669=1093.230,-43.925,-52.321,175.179,15.980,152.383
C08670=1093.224,-44.175,-52.308,175.178,15.978,152.383
C08671=1093.218,-44.424,-52.298,175.176,15.977,152.383
C08672=1093.213,-44.674,-52.285,175.175,15.976,152.383
C08673=1093.207,-44.924,-52.272,175.173,15.975,152.383
C08674=1093.201,-45.174,-52.262,175.171,15.974,152.383
C08675=1093.195,-45.423,-52.249,175.170,15.973,152.383
C08676=1093.189,-45.672,-52.237,175.168,15.972,152.383
C08677=1093.183,-45.922,-52.225,175.166,15.971,152.384
C08678=1093.177,-46.173,-52.213,175.164,15.970,152.384
C08679=1093.171,-46.422,-52.201,175.163,15.969,152.384
C08680=1093.166,-46.671,-52.189,175.161,15.968,152.384
C08681=1093.160,-46.921,-52.178,175.160,15.967,152.384
C08682=1093.154,-47.171,-52.165,175.158,15.966,152.384
C08683=1093.148,-47.420,-52.154,175.156,15.965,152.384
C08684=1093.142,-47.670,-52.142,175.155,15.964,152.385
C08685=1093.136,-47.920,-52.130,175.153,15.963,152.385
C08686=1093.130,-48.169,-52.118,175.151,15.961,152.385
C08687=1093.124,-48.438,-52.105,175.149,15.960,152.385
C08688=1093.117,-48.708,-52.092,175.147,15.959,152.385
C08689=1093.111,-48.977,-52.080,175.145,15.958,152.385
C08690=1093.105,-49.247,-52.067,175.144,15.957,152.385
C08691=1093.099,-49.497,-52.056,175.142,15.956,152.385
C08692=1093.093,-49.746,-52.043,175.140,15.955,152.386
C08693=1093.088,-49.997,-52.032,175.139,15.954,152.386
C08694=1093.082,-50.245,-52.020,175.137,15.953,152.386
C08695=1093.076,-50.495,-52.007,175.136,15.951,152.386
C08696=1093.070,-50.745,-51.997,175.134,15.951,152.386
C08697=1093.063,-50.994,-51.985,175.132,15.950,152.386
C08698=1093.057,-51.245,-51.973,175.130,15.948,152.387
C08699=1093.052,-51.494,-51.961,175.129,15.947,152.387
C08700=1093.045,-51.744,-51.950,175.127,15.947,152.387
C08701=1093.039,-51.993,-51.938,175.125,15.945,152.387
C08702=1093.033,-52.243,-51.926,175.124,15.944,152.387
C08703=1093.028,-52.492,-51.915,175.122,15.944,152.387
C08704=1093.021,-52.742,-51.903,175.120,15.942,152.387
C08705=1093.015,-52.992,-51.891,175.119,15.941,152.388
C08706=1093.009,-53.241,-51.879,175.117,15.941,152.388
C08707=1093.003,-53.491,-51.868,175.115,15.939,152.388
C08708=1092.997,-53.740,-51.857,175.114,15.938,152.388
C08709=1092.991,-53.991,-51.845,175.112,15.938,152.388
C08710=1092.985,-54.240,-51.833,175.110,15.937,152.388
C08711=1092.979,-54.490,-51.822,175.108,15.935,152.388
C08712=1092.972,-54.739,-51.810,175.107,15.935,152.389
C08713=1092.967,-54.989,-51.799,175.105,15.934,152.389
C08714=1092.961,-55.239,-51.787,175.103,15.932,152.389
C08715=1092.955,-55.488,-51.776,175.101,15.932,152.389
C08716=1092.949,-55.738,-51.764,175.100,15.931,152.389
C08717=1092.943,-55.988,-51.752,175.098,15.929,152.389
C08718=1092.937,-56.238,-51.741,175.096,15.929,152.390
C08719=1092.931,-56.487,-51.729,175.095,15.928,152.390
C08720=1092.925,-56.737,-51.718,175.093,15.926,152.390
C08721=1092.919,-56.986,-51.706,175.091,15.926,152.390
C08722=1092.913,-57.236,-51.695,175.090,15.925,152.390
C08723=1092.907,-57.486,-51.684,175.088,15.923,152.390
C08724=1092.901,-57.735,-51.672,175.086,15.922,152.390
C08725=1092.896,-57.985,-51.660,175.085,15.922,152.391
C08726=1092.889,-58.235,-51.649,175.084,15.921,152.391
C08727=1092.883,-58.484,-51.638,175.082,15.920,152.391
C08728=1092.877,-58.734,-51.626,175.080,15.919,152.391
C08729=1092.871,-58.983,-51.615,175.079,15.918,152.391
C08730=1092.865,-59.234,-51.603,175.077,15.917,152.391
C08731=1092.860,-59.483,-51.592,175.075,15.916,152.392
C08732=1092.853,-59.733,-51.580,175.074,15.915,152.392
C08733=1092.847,-59.982,-51.569,175.072,15.914,152.392
C08734=1092.841,-60.232,-51.558,175.070,15.913,152.392
C08735=1092.835,-60.482,-51.546,175.068,15.912,152.392
C08736=1092.830,-60.731,-51.535,175.067,15.911,152.392
C08737=1092.823,-60.981,-51.524,175.065,15.910,152.393
C08738=1092.817,-61.230,-51.512,175.063,15.909,152.393
C08739=1092.811,-61.480,-51.501,175.062,15.908,152.393
C08740=1092.805,-61.730,-51.490,175.060,15.907,152.393
C08741=1092.800,-61.980,-51.478,175.058,15.906,152.393
C08742=1092.794,-62.229,-51.467,175.057,15.905,152.393
C08743=1092.788,-62.479,-51.456,175.055,15.904,152.394
C08744=1092.782,-62.729,-51.444,175.053,15.903,152.394
C08745=1092.776,-62.978,-51.434,175.052,15.903,152.394
C08746=1092.769,-63.228,-51.422,175.050,15.902,152.394
C08747=1092.764,-63.478,-51.410,175.049,15.901,152.394
C08748=1092.758,-63.727,-51.399,175.047,15.900,152.394
C08749=1092.752,-63.977,-51.388,175.045,15.899,152.394
C08750=1092.746,-64.226,-51.376,175.044,15.898,152.395
C08751=1092.740,-64.498,-51.365,175.042,15.897,152.395
C08752=1092.733,-64.768,-51.352,175.040,15.896,152.395
C08753=1092.727,-65.039,-51.340,175.039,15.895,152.395
C08754=1092.720,-65.309,-51.328,175.036,15.893,152.395
C08755=1092.714,-65.560,-51.317,175.035,15.893,152.395
C08756=1092.708,-65.809,-51.306,175.034,15.892,152.395
C08757=1092.703,-66.059,-51.295,175.032,15.891,152.396
C08758=1092.696,-66.309,-51.284,175.030,15.890,152.396
C08759=1092.691,-66.558,-51.271,175.028,15.889,152.396
C08760=1092.685,-66.808,-51.260,175.027,15.888,152.396
C08761=1092.679,-67.058,-51.249,175.025,15.887,152.396
C08762=1092.673,-67.307,-51.238,175.023,15.886,152.396
C08763=1092.667,-67.557,-51.227,175.022,15.885,152.397
C08764=1092.661,-67.807,-51.216,175.020,15.884,152.397
C08765=1092.655,-68.056,-51.205,175.018,15.883,152.397
C08766=1092.649,-68.306,-51.193,175.017,15.882,152.397
C08767=1092.643,-68.555,-51.183,175.016,15.882,152.397
C08768=1092.637,-68.805,-51.172,175.014,15.881,152.397
C08769=1092.632,-69.055,-51.160,175.012,15.880,152.398
C08770=1092.626,-69.305,-51.149,175.010,15.879,152.398
C08771=1092.620,-69.554,-51.138,175.009,15.878,152.398
C08772=1092.614,-69.804,-51.127,175.007,15.877,152.398
C08773=1092.608,-70.054,-51.116,175.005,15.876,152.398
C08774=1092.602,-70.304,-51.105,175.004,15.875,152.398
C08775=1092.597,-70.553,-51.094,175.002,15.874,152.399
C08776=1092.590,-70.803,-51.083,175.000,15.873,152.399
C08777=1092.585,-71.053,-51.072,174.999,15.872,152.399
C08778=1092.579,-71.302,-51.061,174.998,15.872,152.399
C08779=1092.573,-71.552,-51.050,174.996,15.870,152.399
C08780=1092.567,-71.802,-51.039,174.994,15.869,152.399
C08781=1092.561,-72.051,-51.028,174.992,15.869,152.399
C08782=1092.555,-72.301,-51.017,174.991,15.867,152.400
C08783=1092.550,-72.550,-51.006,174.989,15.866,152.400
C08784=1092.543,-72.801,-50.995,174.987,15.866,152.400
C08785=1092.537,-73.050,-50.984,174.986,15.865,152.400
C08786=1092.532,-73.299,-50.973,174.985,15.864,152.400
C08787=1092.526,-73.549,-50.963,174.983,15.863,152.400
C08788=1092.520,-73.799,-50.951,174.981,15.862,152.400
C08789=1092.515,-74.049,-50.940,174.980,15.861,152.401
C08790=1092.508,-74.298,-50.930,174.978,15.860,152.401
C08791=1092.502,-74.548,-50.919,174.976,15.859,152.401
C08792=1092.496,-74.798,-50.907,174.974,15.858,152.401
C08793=1092.490,-75.047,-50.897,174.973,15.857,152.401
C08794=1092.485,-75.297,-50.886,174.972,15.857,152.401
C08795=1092.478,-75.547,-50.874,174.970,15.856,152.402
C08796=1092.472,-75.796,-50.864,174.968,15.855,152.402
C08797=1092.466,-76.046,-50.853,174.967,15.854,152.402
C08798=1092.460,-76.296,-50.842,174.965,15.854,152.402
C08799=1092.454,-76.546,-50.832,174.963,15.852,152.402
C08800=1092.448,-76.795,-50.821,174.961,15.852,152.403
C08801=1092.443,-77.045,-50.810,174.960,15.851,152.403
C08802=1092.436,-77.295,-50.799,174.959,15.851,152.403
C08803=1092.431,-77.545,-50.788,174.957,15.849,152.403
C08804=1092.424,-77.794,-50.778,174.955,15.848,152.403
C08805=1092.418,-78.043,-50.767,174.953,15.848,152.403
C08806=1092.412,-78.293,-50.756,174.952,15.846,152.404
C08807=1092.407,-78.544,-50.745,174.950,15.846,152.404
C08808=1092.401,-78.793,-50.735,174.949,15.845,152.404
C08809=1092.394,-79.042,-50.724,174.947,15.845,152.404
C08810=1092.388,-79.292,-50.713,174.946,15.843,152.404
C08811=1092.382,-79.542,-50.702,174.944,15.843,152.404
C08812=1092.377,-79.791,-50.691,174.942,15.842,152.405
C08813=1092.371,-80.042,-50.681,174.940,15.841,152.405
C08814=1092.365,-80.291,-50.671,174.939,15.840,152.405
C08815=1092.358,-80.564,-50.659,174.937,15.839,152.405
C08816=1092.351,-80.838,-50.647,174.935,15.838,152.405
C08817=1092.345,-81.110,-50.635,174.933,15.837,152.406
C08818=1092.338,-81.383,-50.623,174.931,15.837,152.406
C08819=1092.332,-81.633,-50.613,174.931,15.836,152.406
C08820=1092.326,-81.882,-50.603,174.929,15.835,152.406
C08821=1092.320,-82.132,-50.592,174.927,15.834,152.406
C08822=1092.314,-82.382,-50.581,174.925,15.834,152.407
C08823=1092.307,-82.631,-50.571,174.924,15.832,152.407
C08824=1092.302,-82.881,-50.560,174.922,15.832,152.407
C08825=1092.295,-83.130,-50.550,174.921,15.832,152.407
C08826=1092.289,-83.381,-50.539,174.919,15.831,152.407
C08827=1092.283,-83.630,-50.528,174.917,15.830,152.408
C08828=1092.277,-83.880,-50.518,174.915,15.829,152.408
C08829=1092.271,-84.129,-50.508,174.914,15.828,152.408
C08830=1092.265,-84.379,-50.496,174.913,15.828,152.408
C08831=1092.259,-84.629,-50.487,174.911,15.827,152.408
C08832=1092.253,-84.879,-50.476,174.909,15.826,152.408
C08833=1092.246,-85.128,-50.466,174.907,15.825,152.409
C08834=1092.241,-85.378,-50.455,174.905,15.824,152.409
C08835=1092.235,-85.628,-50.444,174.905,15.824,152.409
C08836=1092.228,-85.877,-50.434,174.903,15.823,152.409
C08837=1092.223,-86.127,-50.423,174.901,15.822,152.409
C08838=1092.216,-86.377,-50.413,174.899,15.821,152.410
C08839=1092.211,-86.626,-50.403,174.897,15.821,152.410
C08840=1092.205,-86.877,-50.392,174.897,15.820,152.410
C08841=1092.198,-87.126,-50.382,174.895,15.820,152.410
C08842=1092.192,-87.376,-50.371,174.893,15.818,152.410
C08843=1092.186,-87.625,-50.361,174.891,15.818,152.411
C08844=1092.180,-87.875,-50.350,174.889,15.817,152.411
C08845=1092.174,-88.124,-50.340,174.888,15.816,152.411
C08846=1092.168,-88.375,-50.330,174.887,15.816,152.411
C08847=1092.162,-88.624,-50.319,174.885,15.815,152.411
C08848=1092.156,-88.874,-50.309,174.883,15.814,152.411
C08849=1092.150,-89.124,-50.298,174.881,15.813,152.412
C08850=1092.144,-89.373,-50.288,174.880,15.813,152.412
C08851=1092.138,-89.623,-50.278,174.878,15.812,152.412
C08852=1092.132,-89.872,-50.268,174.877,15.811,152.412
C08853=1092.126,-90.123,-50.257,174.875,15.810,152.412
C08854=1092.119,-90.372,-50.247,174.874,15.810,152.413
C08855=1092.114,-90.622,-50.236,174.872,15.809,152.413
C08856=1092.108,-90.872,-50.226,174.870,15.808,152.413
C08857=1092.102,-91.121,-50.215,174.869,15.807,152.413
C08858=1092.096,-91.371,-50.205,174.867,15.807,152.413
C08859=1092.090,-91.620,-50.195,174.866,15.807,152.414
C08860=1092.084,-91.870,-50.185,174.864,15.805,152.414
C08861=1092.078,-92.120,-50.175,174.862,15.805,152.414
C08862=1092.072,-92.370,-50.164,174.860,15.804,152.414
C08863=1092.065,-92.620,-50.154,174.859,15.804,152.414
C08864=1092.060,-92.870,-50.144,174.858,15.803,152.415
C08865=1092.053,-93.119,-50.133,174.856,15.802,152.415
C08866=1092.048,-93.369,-50.123,174.854,15.801,152.415
C08867=1092.042,-93.618,-50.113,174.852,15.800,152.415
C08868=1092.036,-93.868,-50.103,174.851,15.800,152.415
C08869=1092.030,-94.117,-50.092,174.849,15.799,152.416
C08870=1092.024,-94.367,-50.082,174.848,15.799,152.416
C08871=1092.018,-94.617,-50.072,174.846,15.797,152.416
C08872=1092.012,-94.867,-50.062,174.845,15.797,152.416
C08873=1092.006,-95.117,-50.052,174.843,15.797,152.416
C08874=1092.000,-95.366,-50.041,174.841,15.795,152.417
C08875=1091.994,-95.617,-50.031,174.839,15.795,152.417
C08876=1091.988,-95.866,-50.021,174.839,15.794,152.417
C08877=1091.982,-96.116,-50.011,174.837,15.794,152.417
C08878=1091.976,-96.365,-50.000,174.835,15.793,152.417
C08879=1091.969,-96.641,-49.990,174.833,15.792,152.418
C08880=1091.963,-96.915,-49.979,174.831,15.791,152.418
C08881=1091.957,-97.190,-49.967,174.829,15.790,152.418
C08882=1091.950,-97.466,-49.956,174.828,15.790,152.418
C08883=1091.944,-97.716,-49.946,174.827,15.789,152.418
C08884=1091.938,-97.965,-49.936,174.825,15.789,152.419
C08885=1091.932,-98.216,-49.925,174.823,15.788,152.419
C08886=1091.926,-98.466,-49.916,174.822,15.788,152.419
C08887=1091.919,-98.715,-49.905,174.820,15.787,152.419
C08888=1091.913,-98.965,-49.896,174.818,15.786,152.419
C08889=1091.907,-99.214,-49.885,174.816,15.785,152.420
C08890=1091.901,-99.464,-49.875,174.815,15.785,152.420
C08891=1091.895,-99.714,-49.866,174.814,15.784,152.420
C08892=1091.889,-99.963,-49.855,174.812,15.784,152.420
C08893=1091.883,-100.213,-49.845,174.810,15.783,152.421
C08894=1091.877,-100.463,-49.836,174.809,15.783,152.421
C08895=1091.870,-100.712,-49.826,174.807,15.782,152.421
C08896=1091.865,-100.962,-49.815,174.805,15.781,152.421
C08897=1091.859,-101.212,-49.806,174.804,15.781,152.421
C08898=1091.852,-101.462,-49.796,174.802,15.780,152.422
C08899=1091.847,-101.711,-49.785,174.801,15.779,152.422
C08900=1091.841,-101.961,-49.776,174.799,15.778,152.422
C08901=1091.834,-102.211,-49.766,174.798,15.778,152.422
C08902=1091.828,-102.460,-49.756,174.796,15.778,152.423
C08903=1091.822,-102.710,-49.746,174.794,15.777,152.423
C08904=1091.816,-102.960,-49.736,174.793,15.777,152.423
C08905=1091.810,-103.210,-49.727,174.791,15.776,152.423
C08906=1091.804,-103.459,-49.716,174.789,15.775,152.423
C08907=1091.798,-103.709,-49.706,174.788,15.775,152.424
C08908=1091.792,-103.959,-49.697,174.786,15.775,152.424
C08909=1091.786,-104.208,-49.687,174.785,15.773,152.424
C08910=1091.779,-104.458,-49.677,174.783,15.773,152.424
C08911=1091.774,-104.708,-49.667,174.782,15.773,152.424
C08912=1091.768,-104.958,-49.657,174.780,15.772,152.425
C08913=1091.762,-105.207,-49.648,174.778,15.771,152.425
C08914=1091.755,-105.457,-49.638,174.777,15.771,152.425
C08915=1091.750,-105.707,-49.627,174.775,15.770,152.425
C08916=1091.744,-105.956,-49.618,174.773,15.769,152.426
C08917=1091.737,-106.206,-49.608,174.772,15.769,152.426
C08918=1091.731,-106.456,-49.598,174.770,15.769,152.426
C08919=1091.725,-106.706,-49.589,174.769,15.768,152.426
C08920=1091.719,-106.955,-49.578,174.768,15.768,152.426
C08921=1091.713,-107.205,-49.568,174.766,15.767,152.427
C08922=1091.707,-107.455,-49.559,174.764,15.766,152.427
C08923=1091.701,-107.705,-49.549,174.762,15.766,152.427
C08924=1091.695,-107.955,-49.540,174.761,15.765,152.427
C08925=1091.688,-108.204,-49.530,174.759,15.765,152.428
C08926=1091.682,-108.454,-49.521,174.757,15.764,152.428
C08927=1091.676,-108.703,-49.510,174.756,15.764,152.428
C08928=1091.670,-108.953,-49.500,174.754,15.763,152.428
C08929=1091.664,-109.203,-49.491,174.752,15.762,152.429
C08930=1091.658,-109.453,-49.481,174.751,15.762,152.429
C08931=1091.652,-109.703,-49.471,174.749,15.762,152.429
C08932=1091.646,-109.953,-49.462,174.747,15.761,152.429
C08933=1091.639,-110.202,-49.452,174.746,15.761,152.430
C08934=1091.633,-110.452,-49.443,174.744,15.760,152.430
C08935=1091.627,-110.702,-49.433,174.742,15.760,152.430
C08936=1091.621,-110.951,-49.423,174.742,15.759,152.430
C08937=1091.614,-111.201,-49.413,174.740,15.758,152.430
C08938=1091.608,-111.451,-49.404,174.739,15.758,152.431
C08939=1091.602,-111.701,-49.394,174.737,15.758,152.431
C08940=1091.596,-111.950,-49.385,174.735,15.757,152.431
C08941=1091.591,-112.200,-49.374,174.734,15.757,152.431
C08942=1091.585,-112.450,-49.365,174.732,15.756,152.432
C08943=1091.577,-112.718,-49.355,174.730,15.756,152.432
C08944=1091.571,-112.986,-49.345,174.728,15.755,152.432
C08945=1091.564,-113.254,-49.334,174.727,15.755,152.432
C08946=1091.558,-113.521,-49.324,174.725,15.754,152.433
C08947=1091.552,-113.771,-49.315,174.723,15.754,152.433
C08948=1091.546,-114.021,-49.305,174.722,15.754,152.433
C08949=1091.540,-114.271,-49.296,174.720,15.753,152.433
C08950=1091.533,-114.521,-49.286,174.718,15.752,152.434
C08951=1091.527,-114.770,-49.276,174.717,15.752,152.434
C08952=1091.522,-115.020,-49.267,174.715,15.752,152.434
C08953=1091.516,-115.269,-49.258,174.713,15.751,152.435
C08954=1091.509,-115.519,-49.248,174.712,15.751,152.435
C08955=1091.503,-115.769,-49.239,174.710,15.750,152.435
C08956=1091.497,-116.019,-49.229,174.708,15.750,152.435
C08957=1091.491,-116.268,-49.219,174.708,15.749,152.435
C08958=1091.485,-116.518,-49.210,174.706,15.748,152.436
C08959=1091.479,-116.768,-49.200,174.705,15.748,152.436
C08960=1091.472,-117.018,-49.191,174.703,15.748,152.436
C08961=1091.466,-117.268,-49.181,174.701,15.747,152.436
C08962=1091.460,-117.517,-49.172,174.700,15.747,152.437
C08963=1091.455,-117.767,-49.163,174.698,15.746,152.437
C08964=1091.449,-118.017,-49.154,174.697,15.746,152.437
C08965=1091.442,-118.267,-49.144,174.694,15.746,152.437
C08966=1091.435,-118.516,-49.135,174.693,15.745,152.438
C08967=1091.429,-118.766,-49.125,174.691,15.745,152.438
C08968=1091.423,-119.016,-49.116,174.690,15.745,152.438
C08969=1091.417,-119.266,-49.106,174.688,15.744,152.439
C08970=1091.411,-119.515,-49.097,174.687,15.744,152.439
C08971=1091.405,-119.765,-49.087,174.685,15.743,152.439
C08972=1091.399,-120.014,-49.078,174.684,15.743,152.439
C08973=1091.393,-120.265,-49.069,174.682,15.743,152.439
C08974=1091.387,-120.515,-49.060,174.680,15.742,152.440
C08975=1091.380,-120.764,-49.051,174.679,15.742,152.440
C08976=1091.374,-121.014,-49.041,174.677,15.741,152.440
C08977=1091.368,-121.264,-49.031,174.676,15.741,152.440
C08978=1091.362,-121.513,-49.022,174.674,15.740,152.441
C08979=1091.356,-121.763,-49.013,174.672,15.740,152.441
C08980=1091.350,-122.013,-49.004,174.671,15.740,152.441
C08981=1091.344,-122.263,-48.994,174.669,15.739,152.442
C08982=1091.337,-122.512,-48.985,174.668,15.739,152.442
C08983=1091.331,-122.762,-48.976,174.666,15.738,152.442
C08984=1091.325,-123.012,-48.966,174.664,15.738,152.442
C08985=1091.319,-123.262,-48.958,174.662,15.738,152.443
C08986=1091.313,-123.511,-48.948,174.661,15.738,152.443
C08987=1091.307,-123.761,-48.938,174.659,15.737,152.443
C08988=1091.300,-124.011,-48.930,174.658,15.737,152.443
C08989=1091.294,-124.260,-48.920,174.656,15.737,152.444
C08990=1091.288,-124.511,-48.911,174.655,15.736,152.444
C08991=1091.283,-124.760,-48.902,174.653,15.735,152.444
C08992=1091.276,-125.010,-48.892,174.651,15.735,152.444
C08993=1091.270,-125.259,-48.883,174.650,15.735,152.445
C08994=1091.264,-125.510,-48.875,174.648,15.735,152.445
C08995=1091.257,-125.759,-48.865,174.646,15.735,152.445
C08996=1091.251,-126.009,-48.855,174.645,15.734,152.446
C08997=1091.245,-126.258,-48.847,174.643,15.734,152.446
C08998=1091.239,-126.508,-48.838,174.641,15.733,152.446
C08999=1091.233,-126.758,-48.828,174.640,15.733,152.446
C09000=1091.226,-127.008,-48.819,174.638,15.732,152.447
C09001=1091.220,-127.258,-48.810,174.637,15.733,152.447
C09002=1091.215,-127.507,-48.801,174.635,15.732,152.447
C09003=1091.208,-127.767,-48.792,174.634,15.732,152.447
C09004=1091.201,-128.025,-48.782,174.632,15.732,152.448
C09005=1091.198,-128.285,-48.772,174.630,15.730,152.448
C09006=1091.203,-128.541,-48.759,174.630,15.727,152.447
C09007=1090.797,-128.563,-48.878,174.587,15.834,152.477
C09008=1090.791,-128.306,-48.891,174.587,15.837,152.477
C09009=1090.795,-128.047,-48.901,174.589,15.838,152.477
C09010=1090.802,-127.788,-48.911,174.591,15.839,152.477
C09011=1090.807,-127.529,-48.921,174.592,15.839,152.476
C09012=1090.814,-127.280,-48.930,174.594,15.839,152.476
C09013=1090.820,-127.030,-48.938,174.596,15.840,152.476
C09014=1090.826,-126.780,-48.948,174.597,15.840,152.476
C09015=1090.832,-126.531,-48.957,174.599,15.841,152.475
C09016=1090.839,-126.281,-48.966,174.600,15.841,152.475
C09017=1090.845,-126.031,-48.975,174.602,15.841,152.475
C09018=1090.851,-125.781,-48.985,174.603,15.841,152.475
C09019=1090.857,-125.531,-48.994,174.605,15.842,152.474
C09020=1090.864,-125.281,-49.002,174.607,15.842,152.474
C09021=1090.869,-125.032,-49.012,174.608,15.842,152.474
C09022=1090.875,-124.782,-49.021,174.610,15.843,152.474
C09023=1090.882,-124.532,-49.031,174.611,15.843,152.473
C09024=1090.888,-124.282,-49.039,174.613,15.844,152.473
C09025=1090.894,-124.032,-49.049,174.615,15.844,152.473
C09026=1090.901,-123.783,-49.058,174.616,15.844,152.473
C09027=1090.906,-123.534,-49.067,174.618,15.845,152.472
C09028=1090.912,-123.284,-49.077,174.619,15.845,152.472
C09029=1090.919,-123.034,-49.085,174.621,15.846,152.472
C09030=1090.925,-122.784,-49.095,174.623,15.846,152.472
C09031=1090.931,-122.534,-49.104,174.624,15.846,152.471
C09032=1090.937,-122.284,-49.114,174.626,15.847,152.471
C09033=1090.943,-122.035,-49.123,174.627,15.847,152.471
C09034=1090.949,-121.785,-49.132,174.629,15.848,152.471
C09035=1090.955,-121.535,-49.142,174.631,15.848,152.470
C09036=1090.962,-121.285,-49.151,174.632,15.848,152.470
C09037=1090.968,-121.036,-49.160,174.634,15.848,152.470
C09038=1090.974,-120.786,-49.170,174.635,15.849,152.469
C09039=1090.980,-120.537,-49.179,174.637,15.849,152.469
C09040=1090.986,-120.287,-49.188,174.639,15.850,152.469
C09041=1090.992,-120.037,-49.197,174.640,15.850,152.469
C09042=1090.998,-119.787,-49.207,174.642,15.851,152.468
C09043=1091.004,-119.537,-49.216,174.643,15.851,152.468
C09044=1091.011,-119.287,-49.225,174.645,15.851,152.468
C09045=1091.017,-119.038,-49.235,174.647,15.852,152.468
C09046=1091.023,-118.788,-49.245,174.648,15.852,152.468
C09047=1091.029,-118.539,-49.254,174.650,15.853,152.467
C09048=1091.035,-118.289,-49.263,174.651,15.853,152.467
C09049=1091.041,-118.039,-49.273,174.653,15.854,152.467
C09050=1091.047,-117.789,-49.282,174.655,15.854,152.467
C09051=1091.053,-117.539,-49.291,174.656,15.855,152.466
C09052=1091.060,-117.289,-49.301,174.658,15.855,152.466
C09053=1091.066,-117.039,-49.310,174.660,15.856,152.466
C09054=1091.072,-116.790,-49.320,174.661,15.856,152.466
C09055=1091.078,-116.540,-49.330,174.663,15.857,152.465
C09056=1091.084,-116.291,-49.339,174.665,15.857,152.465
C09057=1091.091,-116.041,-49.348,174.666,15.857,152.465
C09058=1091.097,-115.791,-49.357,174.668,15.858,152.465
C09059=1091.103,-115.542,-49.367,174.669,15.858,152.464
C09060=1091.109,-115.292,-49.376,174.671,15.859,152.464
C09061=1091.115,-115.042,-49.386,174.672,15.859,152.464
C09062=1091.121,-114.792,-49.396,174.674,15.859,152.464
C09063=1091.128,-114.542,-49.405,174.676,15.860,152.463
C09064=1091.134,-114.293,-49.415,174.677,15.861,152.463
C09065=1091.140,-114.043,-49.424,174.678,15.861,152.463
C09066=1091.146,-113.793,-49.434,174.680,15.862,152.463
C09067=1091.152,-113.543,-49.443,174.682,15.862,152.462
C09068=1091.158,-113.275,-49.453,174.683,15.862,152.462
C09069=1091.165,-113.007,-49.464,174.685,15.863,152.462
C09070=1091.171,-112.739,-49.474,174.687,15.864,152.462
C09071=1091.178,-112.470,-49.484,174.689,15.864,152.461
C09072=1091.184,-112.221,-49.494,174.690,15.864,152.461
C09073=1091.190,-111.971,-49.503,174.692,15.865,152.461
C09074=1091.196,-111.721,-49.514,174.694,15.866,152.461
C09075=1091.202,-111.471,-49.523,174.695,15.866,152.461
C09076=1091.208,-111.221,-49.533,174.696,15.867,152.460
C09077=1091.214,-110.971,-49.542,174.698,15.868,152.460
C09078=1091.221,-110.722,-49.553,174.699,15.868,152.460
C09079=1091.227,-110.472,-49.562,174.701,15.868,152.460
